# B&R Automation Studio project AcpTrakDemoTemplate
Automation Studio 4.10.3.60 SP; technology packages: mapp 5.18.0, mappControl 5.18.0, mappMotion 5.18.0, mappView 5.18.0

## Configuration Config1

CPU X20CP1685, AutomationRuntime G4.90, Build 4.1.2, Safety 0.0, Vc V4.72.2

### Task classes (Cpu.sw)
```
Cyclic#1 (cycle 800 us, tolerance 0 us):
  TrakCtrl <- Source.TrakCtrl.prg
Cyclic#4:
  MappCtrl <- Source.Infrastructure.MappCtrl.prg
Cyclic#8 (cycle 96000 us, tolerance 29952000 us):
  TrakProduc <- Source.Infrastructure.TrakProduction.prg
  TrakSvg <- Source.Infrastructure.TrakSvg.prg
DataObjects: McAcpSys
NcDataObjects: McDriveLog
Binaries: arsvcreg, udbdef, McAcpDrv, arflatprv, McProfGen, arcoal, TCData, FWRules, McAcpSim, mvLoader, ashwd, Config_1, ashwac, User, sysconf, asfw, arconfig, Config_3, Config_2, iomap, Role, Config_4, Config
Libraries: McBase, McAxis, McAcpTrak, MpBase, operator, runtime, astime, AsIecCon, AsBrStr, AsIODiag, sys_lib, standard, MTData, brsystem, MTTypes, MpAlarmX, MpServer, powerlnk, fileio, arssl, dataobj, aruser
```

### Hardware
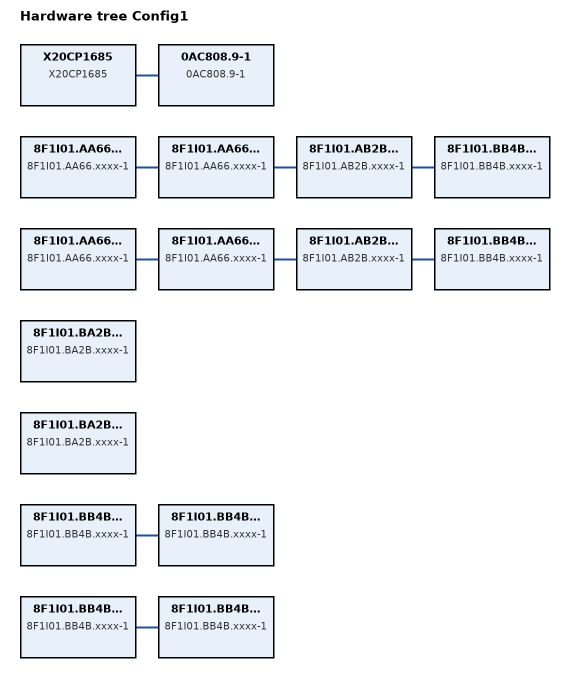
```
0AC808.9-1 : 0AC808.9-1 v1.0.0.0  [ETH1 -> X20CP1685.IF3 [Cable Type=PowerlinkCable, Length=10, Version=1.0.0.3]; ETH5 -> 8F1I01.BB4B.xxxx-1d.PLK3 [Cable Type=PowerlinkCable, Length=10, Version=1.0.0.3]; ETH8 -> 8F1I01.BB4B.xxxx-1e.PLK3 [Cable Type=PowerlinkCable, Length=10, Version=1.0.0.3]]
8F1I01.AA66.xxxx-1 : 8F1I01.AA66.xxxx-1 v1.0.0.2  [PLK1 -> 8F1I01.BA2B.xxxx-1c.PLK2 [Cable Type=PowerlinkCable, Length=10, Version=1.0.0.3]; PLK2 -> 8F1I01.AA66.xxxx-1e.PLK1 [Cable Type=PowerlinkCable, Length=10, Version=1.0.0.3]]
  EnableDNA = on
  DriveConfiguration:
    McTypeID = LLMConfig
  DriveConfiguration/Segment:
    Shape = STRAIGHT660
    SegmentReference = Seg_A_1
    SegmentSectorDirection = Positive
    ElongationCompensation = UseAssemblySetting
    StopReaction = UseAssemblySetting
    SpeedFilter = UseAssemblySetting
8F1I01.AA66.xxxx-1e : 8F1I01.AA66.xxxx-1 v1.0.0.2  [PLK1 -> 8F1I01.AA66.xxxx-1.PLK2 [Cable Type=PowerlinkCable, Length=10, Version=1.0.0.3]; PLK2 -> 8F1I01.AB2B.xxxx-1a.PLK1 [Cable Type=PowerlinkCable, Length=10, Version=1.0.0.3]]
  EnableDNA = on
  DriveConfiguration:
    McTypeID = LLMConfig
  DriveConfiguration/Segment:
    Shape = STRAIGHT660
    SegmentReference = Seg_A_2
    SegmentSectorDirection = Positive
    ElongationCompensation = UseAssemblySetting
    StopReaction = UseAssemblySetting
    SpeedFilter = UseAssemblySetting
8F1I01.AA66.xxxx-1f : 8F1I01.AA66.xxxx-1 v1.0.0.2  [PLK1 -> 8F1I01.BA2B.xxxx-1b.PLK2 [Cable Type=PowerlinkCable, Length=10, Version=1.0.0.3]; PLK2 -> 8F1I01.AA66.xxxx-1k.PLK1 [Cable Type=PowerlinkCable, Length=10, Version=1.0.0.3]]
  EnableDNA = on
  DriveConfiguration:
    McTypeID = LLMConfig
  DriveConfiguration/Segment:
    Shape = STRAIGHT660
    SegmentReference = Seg_A_8
    SegmentSectorDirection = Positive
    ElongationCompensation = UseAssemblySetting
    StopReaction = UseAssemblySetting
    SpeedFilter = UseAssemblySetting
8F1I01.AA66.xxxx-1k : 8F1I01.AA66.xxxx-1 v1.0.0.2  [PLK1 -> 8F1I01.AA66.xxxx-1f.PLK2 [Cable Type=PowerlinkCable, Length=10, Version=1.0.0.3]; PLK2 -> 8F1I01.AB2B.xxxx-1.PLK1 [Cable Type=PowerlinkCable, Length=10, Version=1.0.0.3]]
  EnableDNA = on
  DriveConfiguration:
    McTypeID = LLMConfig
  DriveConfiguration/Segment:
    Shape = STRAIGHT660
    SegmentReference = Seg_A_9
    SegmentSectorDirection = Positive
    ElongationCompensation = UseAssemblySetting
    StopReaction = UseAssemblySetting
    SpeedFilter = UseAssemblySetting
8F1I01.AB2B.xxxx-1 : 8F1I01.AB2B.xxxx-1 v1.0.0.2  [PLK1 -> 8F1I01.AA66.xxxx-1k.PLK2 [Cable Type=PowerlinkCable, Length=10, Version=1.0.0.3]; PLK2 -> 8F1I01.BB4B.xxxx-1.PLK1 [Cable Type=PowerlinkCable, Length=10, Version=1.0.0.3]]
  EnableDNA = on
  DriveConfiguration:
    McTypeID = LLMConfig
  DriveConfiguration/Segment:
    Shape = STRAIGHT105_TO_CIRCULAR
    SegmentReference = Seg_A_10
    SegmentSectorDirection = Positive
    ElongationCompensation = UseAssemblySetting
    StopReaction = UseAssemblySetting
    SpeedFilter = UseAssemblySetting
8F1I01.AB2B.xxxx-1a : 8F1I01.AB2B.xxxx-1 v1.0.0.2  [PLK1 -> 8F1I01.AA66.xxxx-1e.PLK2 [Cable Type=PowerlinkCable, Length=10, Version=1.0.0.3]; PLK2 -> 8F1I01.BB4B.xxxx-1b.PLK1 [Cable Type=PowerlinkCable, Length=10, Version=1.0.0.3]]
  EnableDNA = on
  DriveConfiguration:
    McTypeID = LLMConfig
  DriveConfiguration/Segment:
    Shape = STRAIGHT105_TO_CIRCULAR
    SegmentReference = Seg_A_3
    SegmentSectorDirection = Positive
    ElongationCompensation = UseAssemblySetting
    StopReaction = UseAssemblySetting
    SpeedFilter = UseAssemblySetting
8F1I01.BA2B.xxxx-1b : 8F1I01.BA2B.xxxx-1 v1.0.0.2  [PLK1 -> 8F1I01.BB4B.xxxx-1c.PLK2 [Cable Type=PowerlinkCable, Length=10, Version=1.0.0.3]; PLK2 -> 8F1I01.AA66.xxxx-1f.PLK1 [Cable Type=PowerlinkCable, Length=10, Version=1.0.0.3]]
  EnableDNA = on
  DriveConfiguration:
    McTypeID = LLMConfig
  DriveConfiguration/Segment:
    Shape = CIRCULAR_TO_STRAIGHT105
    SegmentReference = Seg_A_7
    SegmentSectorDirection = Positive
    ElongationCompensation = UseAssemblySetting
    StopReaction = UseAssemblySetting
    SpeedFilter = UseAssemblySetting
8F1I01.BA2B.xxxx-1c : 8F1I01.BA2B.xxxx-1 v1.0.0.2  [PLK1 -> 8F1I01.BB4B.xxxx-1a.PLK2 [Cable Type=PowerlinkCable, Length=10, Version=1.0.0.3]; PLK2 -> 8F1I01.AA66.xxxx-1.PLK1 [Cable Type=PowerlinkCable, Length=10, Version=1.0.0.3]]
  EnableDNA = on
  DriveConfiguration:
    McTypeID = LLMConfig
  DriveConfiguration/Segment:
    Shape = CIRCULAR_TO_STRAIGHT105
    SegmentReference = Seg_A_14
    SegmentSectorDirection = Positive
    ElongationCompensation = UseAssemblySetting
    StopReaction = UseAssemblySetting
    SpeedFilter = UseAssemblySetting
8F1I01.BB4B.xxxx-1 : 8F1I01.BB4B.xxxx-1 v1.0.0.2  [PLK1 -> 8F1I01.AB2B.xxxx-1.PLK2 [Cable Type=PowerlinkCable, Length=10, Version=1.0.0.3]]
  EnableDNA = on
  DriveConfiguration:
    McTypeID = LLMConfig
  DriveConfiguration/Segment:
    Shape = CIRCULAR
    SegmentReference = Seg_A_11
    SegmentSectorDirection = Positive
    ElongationCompensation = UseAssemblySetting
    StopReaction = UseAssemblySetting
    SpeedFilter = UseAssemblySetting
8F1I01.BB4B.xxxx-1a : 8F1I01.BB4B.xxxx-1 v1.0.0.2  [PLK1 -> 8F1I01.BB4B.xxxx-1d.PLK2 [Cable Type=PowerlinkCable, Length=10, Version=1.0.0.3]; PLK2 -> 8F1I01.BA2B.xxxx-1c.PLK1 [Cable Type=PowerlinkCable, Length=10, Version=1.0.0.3]]
  EnableDNA = on
  DriveConfiguration:
    McTypeID = LLMConfig
  DriveConfiguration/Segment:
    Shape = CIRCULAR
    SegmentReference = Seg_A_13
    SegmentSectorDirection = Positive
    ElongationCompensation = UseAssemblySetting
    StopReaction = UseAssemblySetting
    SpeedFilter = UseAssemblySetting
8F1I01.BB4B.xxxx-1b : 8F1I01.BB4B.xxxx-1 v1.0.0.2  [PLK1 -> 8F1I01.AB2B.xxxx-1a.PLK2 [Cable Type=PowerlinkCable, Length=10, Version=1.0.0.3]]
  EnableDNA = on
  DriveConfiguration:
    McTypeID = LLMConfig
  DriveConfiguration/Segment:
    Shape = CIRCULAR
    SegmentReference = Seg_A_4
    SegmentSectorDirection = Positive
    ElongationCompensation = UseAssemblySetting
    StopReaction = UseAssemblySetting
    SpeedFilter = UseAssemblySetting
8F1I01.BB4B.xxxx-1c : 8F1I01.BB4B.xxxx-1 v1.0.0.2  [PLK1 -> 8F1I01.BB4B.xxxx-1e.PLK2 [Cable Type=PowerlinkCable, Length=10, Version=1.0.0.3]; PLK2 -> 8F1I01.BA2B.xxxx-1b.PLK1 [Cable Type=PowerlinkCable, Length=10, Version=1.0.0.3]]
  EnableDNA = on
  DriveConfiguration:
    McTypeID = LLMConfig
  DriveConfiguration/Segment:
    Shape = CIRCULAR
    SegmentReference = Seg_A_6
    SegmentSectorDirection = Positive
    ElongationCompensation = UseAssemblySetting
    StopReaction = UseAssemblySetting
    SpeedFilter = UseAssemblySetting
8F1I01.BB4B.xxxx-1d : 8F1I01.BB4B.xxxx-1 v1.0.0.2  [PLK2 -> 8F1I01.BB4B.xxxx-1a.PLK1 [Cable Type=PowerlinkCable, Length=10, Version=1.0.0.3]; PLK3 -> 0AC808.9-1.ETH5 [Cable Type=PowerlinkCable, Length=10, Version=1.0.0.3]]
  EnableDNA = on
  DriveConfiguration:
    McTypeID = LLMConfig
  DriveConfiguration/Segment:
    Shape = CIRCULAR
    SegmentReference = Seg_A_12
    SegmentSectorDirection = Positive
    ElongationCompensation = UseAssemblySetting
    StopReaction = UseAssemblySetting
    SpeedFilter = UseAssemblySetting
8F1I01.BB4B.xxxx-1e : 8F1I01.BB4B.xxxx-1 v1.0.0.2  [PLK2 -> 8F1I01.BB4B.xxxx-1c.PLK1 [Cable Type=PowerlinkCable, Length=10, Version=1.0.0.3]; PLK3 -> 0AC808.9-1.ETH8 [Cable Type=PowerlinkCable, Length=10, Version=1.0.0.3]]
  EnableDNA = on
  DriveConfiguration:
    McTypeID = LLMConfig
  DriveConfiguration/Segment:
    Shape = CIRCULAR
    SegmentReference = Seg_A_5
    SegmentSectorDirection = Positive
    ElongationCompensation = UseAssemblySetting
    StopReaction = UseAssemblySetting
    SpeedFilter = UseAssemblySetting
X20CP1685 : X20CP1685 v1.4.0.0
  Connector IF2:
    ActivateDevice = 1
  Connector IF3:
    CycleTime = 800
  ConfigurationID = AcpTrakVolpak_Config1
  Simulation = 1
  TimerDeviceType = EPLX2X
  TimerDevice = X20CP1685.IF3
  TaskClassIdleTime = 800
  Cyclic1Duration = 800
  Cyclic1Tolerance = 0
  Cyclic3Duration = 49600
  Cyclic3Tolerance = 49600
  Cyclic8Duration = 96000
  Cyclic8Tolerance = 29952000
  FileDevice1
  FileDeviceName1 = SvgData
  FileDevicePath1 = C:\DataTrak\
  ActivateOpcUa = 1
  OpcUaInformationModels_PV_Version = 1
```

### Config_1.assembly - X20CP1685/mappMotion/TrakOval/Config_1.assembly
```
Element gAssembly_1 (Type=assembly)
  Tracks:
    TrackSeparation = 0.030
    Track[1]:
      Segments:
        SegmentRef[1] = ::Seg_A_1
        SegmentRef[2] = ::Seg_A_2
        SegmentRef[3] = ::Seg_A_3
        SegmentRef[4] = ::Seg_A_4
        SegmentRef[5] = ::Seg_A_5
        SegmentRef[6] = ::Seg_A_6
        SegmentRef[7] = ::Seg_A_7
        SegmentRef[8] = ::Seg_A_8
        SegmentRef[9] = ::Seg_A_9
        SegmentRef[10] = ::Seg_A_10
        SegmentRef[11] = ::Seg_A_11
        SegmentRef[12] = ::Seg_A_12
        SegmentRef[13] = ::Seg_A_13
        SegmentRef[14] = ::Seg_A_14
      Position = Absolute
        SegmentRef = ::Seg_A_1
        SegmentCountDirection = RightToLeft
        Translation:
          X = 0.0
          Y = 0.0
          Z = 0.0
        Orientation:
          Angle1 = 0.0
          Angle2 = 180.0
          Angle3 = 0.0
  CommonSegmentSettings:
    SegmentSimulationOnPLC = Off
    ElongationCompensation = Inactive
    StopReaction = InductionHalt
    SpeedFilter = Lowpass
      FilterTime = 0.0008
    ControllerParameters:
      DefaultParameter:
        Controller:
          Position:
            ProportionalGain = 200
          Speed:
            ProportionalGain = 80
            IntegrationTime = 0.0
          FeedForward:
            TotalMass = 1.0
            ForcePositive = 1.5
            ForceNegative = 1.5
            SpeedForceFactor = 1.4
            ForceLoad = 0.0
        MovementErrorLimits:
          PositionError = 0.01
          VelocityError = 50
        Diverter:
          ForceOverride = 1.0
      AdditionalParameterSets = NotUsed
    ScopeOfErrorReaction = Assembly
    ShuttleIdentificationTime = 0
  Shuttles:
    MaxShuttleCount = 100
    MaxShuttleCommandCount = 0
    UseConvoys = Active
    DistanceReserve:
      Collision = 0.002
      ErrorStop = 0.006
    ShuttleStereotypes:
      ShuttleStRef[1] = ShuttleStereotype_1
    MagnetPlateConfigurations:
      ShuttleType[1] = 8F1SA.102.xxxxxx-x
    CollisionAvoidance:
      Strategy = Constant
      MaximumModelDimensions:
        Length:
          ExtentToFront = 0.025
          ExtentToBack = 0.025
        Width:
          Width = 0.046
  Visualization:
    MonitoringPv = 
    ProcessingTaskClass = 4
  Alarms = MpAlarmX
```

### Config_2.shuttlestereotype - X20CP1685/mappMotion/TrakOval/Config_2.shuttlestereotype
```
Element ShuttleStereotype_1 (Type=shuttlestereotype)
  MeasurementUnit = 5067858
  MeasurementResolution = 0.00001
  MovementLimits = Internal
    VelocityIsReadOnly = 0
    Velocity:
      Velocity = 4.0
    AccelerationIsReadOnly = 0
    Acceleration:
      Acceleration = 40.0
    DecelerationIsReadOnly = 0
    Deceleration:
      Deceleration = 40.0
    UpdateMode = Immediately
  JerkFilter = NotUsed
  UserData:
    Size = 52
  StateTransitions:
    AutomaticRecontrol = Active
```

### Config_3.sector - X20CP1685/mappMotion/TrakOval/Config_3.sector
```
Element SectorTrackA (Type=sector)
  Type = Composed
    StartSegment:
      SegmentRef = ::Seg_A_1
    IntermediateSegments:
      SegmentRef[1] = ::Seg_A_1
      SegmentRef[2] = ::Seg_A_2
      SegmentRef[3] = ::Seg_A_3
      SegmentRef[4] = ::Seg_A_4
      SegmentRef[5] = ::Seg_A_5
      SegmentRef[6] = ::Seg_A_6
      SegmentRef[7] = ::Seg_A_7
      SegmentRef[8] = ::Seg_A_8
      SegmentRef[9] = ::Seg_A_9
      SegmentRef[10] = ::Seg_A_10
      SegmentRef[11] = ::Seg_A_11
      SegmentRef[12] = ::Seg_A_12
      SegmentRef[13] = ::Seg_A_13
    EndSegment:
      SegmentRef = ::Seg_A_14
      PositionRelativeTo = FromEnd
  Alarms = MpAlarmX
```

### Config_4.processpointlist - X20CP1685/mappMotion/TrakOval/Config_4.processpointlist
```
Element ProcessPointList_Template (Type=processpointlist)
  ProcessPoint[0]:
    Name = PP_Test
    SectorRef = SectorTrackA
    TriggerEventBufferSize = 10
    BarrierFunctionality = Off
Element ProcessPointList_Machine (Type=processpointlist)
  ProcessPoint[0]:
    Name = PP_Init
    SectorRef = SectorTrackA
    TriggerEventBufferSize = 10
    BarrierFunctionality = On
  ProcessPoint[1]:
    Name = PP_Stop
    SectorRef = SectorTrackA
    Position = 1.5
    TriggerEventBufferSize = 10
    BarrierFunctionality = On
  ProcessPoint[2]:
    Name = PP_Stop1
    SectorRef = SectorTrackA
    Position = 3
    TriggerEventBufferSize = 10
    BarrierFunctionality = On
```

### Config_5.mappmotioncfg - X20CP1685/mappMotion/TrakOval/Config_5.mappmotioncfg
```
Element MappMotionConfiguration (Type=mappmotioncfg)
  Processing:
    ProcessingTaskClass = 1
  SharedAlarms:
    Axis = MpAlarmX
    Segment = MpAlarmX
    Sector = MpAlarmX
    Shuttle = MpAlarmX
      mapp.AlarmX.Core.Configuration:
        [3]:
          AdditionalInformation1 = Shuttle
```

## Logical view

Binary libraries used (declarations not repeated): operator, runtime, astime, AsIecCon, AsBrStr, AsIODiag, sys_lib, standard, McBase, McAcpTrak, McAxis, MpBase, MTData 5.18.0, brsystem, MTTypes, MpAlarmX, MpServer

### Global.var
```iecst
VAR
	Seg_A_1 : McSegmentType;
	Seg_A_2 : McSegmentType;
	Seg_A_3 : McSegmentType;
	Seg_A_4 : McSegmentType;
	Seg_A_5 : McSegmentType;
	Seg_A_6 : McSegmentType;
	Seg_A_7 : McSegmentType;
	Seg_A_8 : McSegmentType;
	Seg_A_9 : McSegmentType;
	Seg_A_10 : McSegmentType;
	Seg_A_11 : McSegmentType;
	Seg_A_12 : McSegmentType;
	Seg_A_13 : McSegmentType;
	Seg_A_14 : McSegmentType;
END_VAR
```

### gTrak.typ - Global data types
```iecst
(*interface assembly control*)

TYPE
	TrakAsmType : 	STRUCT
		AssemblyRef : REFERENCE TO McAssemblyType; (*assembly reference - ADR(gAssembly_1)*)
		CmdPower : BOOL; (*command power on/off*)
		CmdErrorReset : BOOL; (*command error reset*)
		CmdAllShuttleMoveStop : BOOL;
		CmdAllShuttleMovePosition : BOOL;
		CmdAllShuttleMoveVelocity : BOOL;
		StatusSimulated : BOOL; (*status assembly is simulated*)
		StatusDisabled : BOOL; (*status assembly is disabled*)
		StatusReady : BOOL; (*status assembly is ready*)
		StatusHoming : BOOL; (*status assembly is homing*)
		StatusStopping : BOOL; (*status assembly is stopping*)
		StatusErrorStop : BOOL; (*status assembly is in error-stop*)
		StatusCommunicationReady : BOOL; (*status PLK communication to all segments in assembly is ready*)
		StatusReadyForPower : BOOL; (*status assembly is ready for command power-on*)
		StatusPower : BOOL; (*status assembly is power-on*)
		StatusReadyForMovement : BOOL; (*status assembly is ready to start shuttle movements*)
		MonitorSegmentsPresent : UINT; (*monitor segment present on assembly*)
		MonitorSegmentsInErrorStop : UINT; (*monitor segment in error-stop*)
		MonitorShuttlesPresent : UINT; (*monitor shuttles present on assembly*)
		MonitorShuttlesInErrorStop : UINT; (*monitor shuttles in error-stop*)
		ParaMoveSectorRef : REFERENCE TO McSectorType; (*parameter shuttle move target sector - ADR(Sector_x)*)
		ParaMovePosition : LREAL; (*parameter shuttle move target position*)
		ParaMoveVelocity : REAL; (*parameter shuttle move target velocity*)
		ParaMoveRouteVelocity : REAL; (*parameter shuttle move routing velocity*)
		ParaMoveAcceleration : REAL; (*parameter shuttle move acceleration*)
		ParaMoveDeceleration : REAL; (*parameter shuttle move deceleration*)
		Segment : ARRAY[1..TRAK_MAX_SEGMENT]OF TrakAsmSegmentType;
		Shuttle : ARRAY[1..TRAK_MAX_SHUTTLE]OF TrakAsmShuttleType; (*shuttle information*)
	END_STRUCT;
	TrakAsmShuttleType : 	STRUCT
		Valid : BOOL; (*shuttledata valid*)
		Axis : McAxisType; (*McAxis of shuttle*)
		ID : UDINT; (*shuttle ID as displayed in logger and SceneViewer - TODO*)
		ActSectorType : McAcpTrakSecTypeEnum; (*shuttle current sector type*)
		ActSector : STRING[32]; (*shuttle current sector*)
		ActPosition : LREAL; (*shuttle position on sector*)
		ActVelocity : REAL; (*shuttle velocity on sector*)
		TotalMoveDistance : LREAL; (*shuttle total moved distance*)
		StatusStandStill : BOOL; (*shuttle is in state Standstill*)
		StatusStopping : BOOL; (*shuttle is in state Stopping*)
		StatusErrorStop : BOOL; (*shuttle is in state Errorstop*)
		StatusDiscreteMotion : BOOL; (*shuttle is in state DiscreteMotion*)
		StatusContinuousMotion : BOOL; (*shuttle is in state ContinuousMotion*)
		StatusSynchronizedMotion : BOOL; (*shuttle is in state SynchronizedMotion*)
	END_STRUCT;
	TrakAsmSegmentType : 	STRUCT
		Valid : BOOL;
		Segment : McSegmentType;
		StatusDisabled : BOOL;
		StatusReady : BOOL;
		StatusStopping : BOOL;
		StatusErrorStop : BOOL;
		StatusShuttlesInError : BOOL;
	END_STRUCT;
END_TYPE

(*shuttle UserData structure - adapt to your application*)

TYPE
	TrakShuttleUserDataType : 	STRUCT
		SceneColorRed : REAL; (*do not change: SceneViewer shuttle colour red*)
		SceneColorGreen : REAL; (*do not change: SceneViewer shuttle colour green*)
		SceneColorBlue : REAL; (*do not change: SceneViewer shuttle colour blue*)
		SceneText : STRING[31]; (*do not change: SceneViewer shuttle text*)
		Test : USINT; (*do not change: for use in TrakTest task*)
		ID : UINT; (*shuttle ID*)
		InitDone : BOOL; (*example: product weight*)
	END_STRUCT;
END_TYPE
```

### gTrak.var - Global variables
```iecst
(*interface assembly control*)
VAR
	gTrakAsm : TrakAsmType; (*trak assembly main interface structure*)
END_VAR
(*production control*)
VAR
	gProducedProduct : UINT; (*number of produced products (in ppm)*)
END_VAR
(*constants*)
VAR CONSTANT
	TRAK_MAX_SHUTTLE : UINT := 72; (*maximum number of shuttles handled in this application - should be set equal or higher than Shuttles-maximum-count setting in mappMotion assembly config file*)
	TRAK_MAX_SEGMENT : UINT := 24; (*maximum number of segments handled in this application*)
END_VAR
```

### Program Logical/Source/TrakCtrl (IEC) - trak assembly control

#### Types.typ
```iecst
(*enum*)

TYPE
	TrakSimShuttleType : 	STRUCT
		SectorRef : REFERENCE TO McSectorType; (*add shuttle in simulation at sector - ADR(Sector_x)*)
		Position : LREAL; (*add shuttle in simulation at position*)
	END_STRUCT;
	StepEnum :
		(
		COMMAND := 0,
		RESET,
		ASM_POWER_ON := 10,
		ASM_POWER_ON_WAIT,
		GET_SEGMENT_INIT := 20,
		GET_SEGMENT,
		GET_SEGMENT_WAIT,
		ADD_SHUTTLE_INIT := 30,
		ADD_SHUTTLE,
		ADD_SHUTTLE_WAIT,
		GET_SHUTTLE_INIT := 40,
		GET_SHUTTLE,
		GET_SHUTTLE_WAIT,
		ERROR := 99,
		READY := 100,
		ASM_POWER_OFF := 110,
		ASM_POWER_OFF_WAIT,
		ASM_SH_DELETE,
		ASM_SH_DELETE_WAIT,
		STOP_SHUTTLE := 120,
		STOP_SHUTTLE_WAIT,
		MOVE_SHUTTLE_VELOCITY := 130,
		MOVE_SHUTTLE_VELOCITY_WAIT,
		MOVE_SHUTTLE_POSITION := 140,
		MOVE_SHUTTLE_POSITION_WAIT
		);
END_TYPE
```

#### Variables.var
```iecst
(*sequence control*)
VAR
	Step : StepEnum;
	i : UINT;
	CntShuttle : UINT;
	CntSegment : UINT;
END_VAR
(*add shuttles for simulation*)
VAR
	SimNumShuttle : USINT := 4;
	SimShuttle : ARRAY[1..TRAK_MAX_SHUTTLE] OF TrakSimShuttleType;
END_VAR
(*initialze shuttle user data*)
VAR
	SizeofShuttleUserData : UDINT;
	ShuttleUserData : TrakShuttleUserDataType;
END_VAR
(*assembly FUB*)
VAR
	MC_BR_AsmReset_AcpTrak_0 : MC_BR_AsmReset_AcpTrak;
	MC_BR_AsmPowerOn_AcpTrak_0 : MC_BR_AsmPowerOn_AcpTrak;
	MC_BR_AsmPowerOff_AcpTrak_0 : MC_BR_AsmPowerOff_AcpTrak;
	MC_BR_AsmGetInfo_AcpTrak_0 : MC_BR_AsmGetInfo_AcpTrak;
	MC_BR_AsmReadStatus_AcpTrak_0 : MC_BR_AsmReadStatus_AcpTrak;
	MC_BR_AsmReadInfo_AcpTrak_0 : MC_BR_AsmReadInfo_AcpTrak;
	MC_BR_AsmGetSegment_AcpTrak_0 : MC_BR_AsmGetSegment_AcpTrak;
	MC_BR_SecAddShuttle_AcpTrak_0 : MC_BR_SecAddShuttle_AcpTrak;
	MC_BR_AsmGetShuttle_AcpTrak_0 : MC_BR_AsmGetShuttle_AcpTrak;
	MC_BR_AsmDeleteShuttle_AcpTrak_0 : MC_BR_AsmDeleteShuttle_AcpTrak;
END_VAR
(*segment FUB*)
VAR
	MC_BR_SegReadStatus_AcpTrak_0 : ARRAY[1..TRAK_MAX_SEGMENT] OF MC_BR_SegReadStatus_AcpTrak;
END_VAR
(*shuttle FUB*)
VAR
	MC_BR_ShCopyUserData_AcpTrak_0 : MC_BR_ShCopyUserData_AcpTrak;
	MC_BR_ShReadInfo_AcpTrak_0 : ARRAY[1..TRAK_MAX_SHUTTLE] OF MC_BR_ShReadInfo_AcpTrak;
	MC_ReadStatus_0 : ARRAY[1..TRAK_MAX_SHUTTLE] OF MC_ReadStatus;
	MC_Stop_0 : MC_Stop;
	MC_BR_RoutedMoveVel_AcpTrak_0 : MC_BR_RoutedMoveVel_AcpTrak;
	MC_BR_RoutedMoveAbs_AcpTrak_0 : MC_BR_RoutedMoveAbs_AcpTrak;
END_VAR
```

#### Main.st
```iecst
//////////////////////////////////////////////////////////////////////////////////////////////////////////////////////////////
//
// Copyright B&R Industrial Automation GmbH
// Author    B&R
// Created   Feb 1, 2018
//
// trak assembly basic control task
// TC#1 => preferred to be attached to mappMotion task class
//
// * assembly startup sequence
// * ErrorStop handling
// * basic shuttle handling
// * aggregated shuttle move commands
//
// "gTrakAsm" - global interface structure
//
//////////////////////////////////////////////////////////////////////////////////////////////////////////////////////////////

PROGRAM _INIT

	//////////////////////////////////////////////////////////////////////////////////////////////////////////////////////////////
	// interface structure

	gTrakAsm.AssemblyRef				:= ADR(gAssembly_1);
	gTrakAsm.CmdPower					:= FALSE;
	gTrakAsm.CmdErrorReset				:= FALSE;

	gTrakAsm.CmdAllShuttleMoveStop		:= FALSE;
	gTrakAsm.CmdAllShuttleMovePosition	:= FALSE;
	gTrakAsm.CmdAllShuttleMoveVelocity	:= FALSE;
	gTrakAsm.ParaMoveSectorRef			:= ADR(SectorTrackA);
	gTrakAsm.ParaMovePosition			:= 2.0;
	gTrakAsm.ParaMoveVelocity			:= 2.0;
	gTrakAsm.ParaMoveRouteVelocity		:= 2.0;
	gTrakAsm.ParaMoveAcceleration		:= 20.0;
	gTrakAsm.ParaMoveDeceleration		:= 20.0;

	Step := COMMAND;

	// size of ShuttleUserData structure - this value has to be entered in ShuttleStereotype -> UserData -> Size
	SizeofShuttleUserData := SIZEOF(ShuttleUserData);

END_PROGRAM

PROGRAM _CYCLIC

	//////////////////////////////////////////////////////////////////////////////////////////////////////////////////////////////
	// global ErrorStop and ErrorReset
	IF(gTrakAsm.StatusErrorStop)THEN
		gTrakAsm.StatusReadyForMovement := FALSE;
		Step := ERROR;
	END_IF
	IF(gTrakAsm.CmdErrorReset)THEN
		gTrakAsm.CmdErrorReset := FALSE;
		MC_BR_AsmReset_AcpTrak_0.Execute := TRUE;
	END_IF

	CASE Step OF

		//////////////////////////////////////////////////////////////////////////////////////////////////////////////////////////////
		// command
		COMMAND:
			IF(gTrakAsm.CmdPower)THEN
				Step := RESET;
			END_IF

		//////////////////////////////////////////////////////////////////////////////////////////////////////////////////////////////
		// startup sequence

		// reset
		RESET:

			brsmemset(ADR(gTrakAsm.Segment), 0, SIZEOF(gTrakAsm.Segment));
			brsmemset(ADR(gTrakAsm.Shuttle), 0, SIZEOF(gTrakAsm.Shuttle));

			MC_BR_AsmGetSegment_AcpTrak_0.Enable := FALSE;
			MC_BR_AsmGetShuttle_AcpTrak_0.Enable := FALSE;

			Step := ASM_POWER_ON;

		// assembly power ON
		ASM_POWER_ON:

			IF(gTrakAsm.StatusDisabled)THEN
				MC_BR_AsmPowerOn_AcpTrak_0.Execute := TRUE;
			END_IF
			Step := ASM_POWER_ON_WAIT;

		ASM_POWER_ON_WAIT:

			IF(gTrakAsm.StatusReady)THEN
				Step := GET_SEGMENT_INIT;
			END_IF

		GET_SEGMENT_INIT:

			MC_BR_AsmGetSegment_AcpTrak_0.Enable 	:= TRUE;
			MC_BR_AsmGetSegment_AcpTrak_0.Next 		:= FALSE;
			CntSegment 	:= 0;
			Step 		:= GET_SEGMENT_WAIT;

		GET_SEGMENT:

			MC_BR_AsmGetSegment_AcpTrak_0.Next := TRUE;
			Step := GET_SEGMENT_WAIT;

		GET_SEGMENT_WAIT:

			IF(MC_BR_AsmGetSegment_AcpTrak_0.Error)THEN
				MC_BR_AsmGetSegment_AcpTrak_0.Enable := FALSE;
				Step := ERROR;

			ELSIF (MC_BR_AsmGetSegment_AcpTrak_0.Valid) THEN

				gTrakAsm.MonitorSegmentsPresent := MC_BR_AsmGetSegment_AcpTrak_0.TotalCount;

				IF(MC_BR_AsmGetSegment_AcpTrak_0.TotalCount = 0)THEN	// no segments present present
					MC_BR_AsmGetSegment_AcpTrak_0.Enable := FALSE;
					Step := ERROR;
				ELSE

					CntSegment := CntSegment + 1;
					gTrakAsm.Segment[CntSegment].Segment := MC_BR_AsmGetSegment_AcpTrak_0.Segment;

					IF(MC_BR_AsmGetSegment_AcpTrak_0.RemainingCount = 0)THEN	// all present segments read => ok, proceed
						MC_BR_AsmGetSegment_AcpTrak_0.Enable := FALSE;
						Step := ADD_SHUTTLE_INIT;
					ELSIF(CntSegment >= TRAK_MAX_SEGMENT)THEN					// more segments present than max configured => error
						MC_BR_AsmGetSegment_AcpTrak_0.Enable := FALSE;
						Step := ERROR;
					ELSE														// read next => positive edge on .Next flag
						MC_BR_AsmGetSegment_AcpTrak_0.Next := FALSE;
						Step := GET_SEGMENT;
					END_IF
				END_IF

			END_IF

		// add shuttles (for simulation only)
		ADD_SHUTTLE_INIT:

			IF(gTrakAsm.StatusSimulated)THEN
				// Define the simulated position for each shuttle
				FOR i:=1 TO TRAK_MAX_SHUTTLE DO
					IF ((i < SimNumShuttle) AND (SimNumShuttle <= TRAK_MAX_SHUTTLE)) THEN
						SimShuttle[i].SectorRef := ADR(SectorTrackA);
						SimShuttle[i].Position 	:= 0.355 + UINT_TO_LREAL(SimNumShuttle - i)/10.0;
					ELSE
						SimShuttle[i].SectorRef := ADR(SectorTrackA);
						SimShuttle[i].Position 	:= 0.355;
					END_IF
				END_FOR
				CntShuttle 	:= 0;
				Step 		:= ADD_SHUTTLE;
			ELSE
				Step := GET_SHUTTLE_INIT;
			END_IF

		ADD_SHUTTLE:

			CntShuttle := CntShuttle + 1;
			IF(CntShuttle > SimNumShuttle)THEN
				Step := GET_SHUTTLE_INIT;
			ELSIF(SimShuttle[CntShuttle].SectorRef = 0)THEN
				Step := GET_SHUTTLE_INIT;
			ELSE
				MC_BR_SecAddShuttle_AcpTrak_0.Sector		:= SimShuttle[CntShuttle].SectorRef;
				MC_BR_SecAddShuttle_AcpTrak_0.Execute		:= TRUE;
				MC_BR_SecAddShuttle_AcpTrak_0.Position		:= SimShuttle[CntShuttle].Position;
				MC_BR_SecAddShuttle_AcpTrak_0.AdvancedParameters.Velocity		:= 0.0;
				MC_BR_SecAddShuttle_AcpTrak_0.AdvancedParameters.Orientation	:= mcDIR_POSITIVE;
				Step := ADD_SHUTTLE_WAIT;
			END_IF

		ADD_SHUTTLE_WAIT:
			IF(MC_BR_SecAddShuttle_AcpTrak_0.Error)THEN
				Step := ERROR;

			ELSIF(MC_BR_SecAddShuttle_AcpTrak_0.Done)THEN
				Step := ADD_SHUTTLE;
			END_IF

		// get all shuttles present on assembly
		GET_SHUTTLE_INIT:

			MC_BR_AsmGetShuttle_AcpTrak_0.Enable 	:= TRUE;
			MC_BR_AsmGetShuttle_AcpTrak_0.Next 		:= FALSE;
			CntShuttle 	:= 0;
			Step 		:= GET_SHUTTLE_WAIT;

		GET_SHUTTLE:

			MC_BR_AsmGetShuttle_AcpTrak_0.Next := TRUE;
			Step := GET_SHUTTLE_WAIT;

		GET_SHUTTLE_WAIT:

			IF(MC_BR_AsmGetShuttle_AcpTrak_0.Error)THEN
				MC_BR_AsmGetShuttle_AcpTrak_0.Enable := FALSE;
				Step := ERROR;

			ELSIF(MC_BR_AsmGetShuttle_AcpTrak_0.Valid)THEN
				gTrakAsm.MonitorShuttlesPresent := MC_BR_AsmGetShuttle_AcpTrak_0.TotalCount;

				IF(MC_BR_AsmGetShuttle_AcpTrak_0.TotalCount = 0)THEN			// no shuttles present => ok, proceed
					MC_BR_AsmGetShuttle_AcpTrak_0.Enable := FALSE;
					Step := READY;
				ELSE
					CntShuttle := CntShuttle + 1;
					gTrakAsm.Shuttle[CntShuttle].Axis	:= MC_BR_AsmGetShuttle_AcpTrak_0.Axis;
					gTrakAsm.Shuttle[CntShuttle].ID		:= MC_BR_AsmGetShuttle_AcpTrak_0.AdditionalInfo.ShuttleID;

					// initialize shuttle UserData (White colour)
					ShuttleUserData.SceneColorRed	:= 1.0;
					ShuttleUserData.SceneColorGreen	:= 1.0;
					ShuttleUserData.SceneColorBlue	:= 1.0;
					ShuttleUserData.ID				:= CntShuttle;

					MC_BR_ShCopyUserData_AcpTrak_0.Axis			:= ADR(gTrakAsm.Shuttle[CntShuttle].Axis);
					MC_BR_ShCopyUserData_AcpTrak_0.Execute		:= TRUE;
					MC_BR_ShCopyUserData_AcpTrak_0.DataAddress	:= ADR(ShuttleUserData);
					MC_BR_ShCopyUserData_AcpTrak_0.DataSize		:= SIZEOF(ShuttleUserData);
					MC_BR_ShCopyUserData_AcpTrak_0.Mode			:= mcACPTRAK_USERDATA_SET;

					IF(MC_BR_AsmGetShuttle_AcpTrak_0.RemainingCount = 0)THEN	// all present shuttles read => ok, proceed
						MC_BR_AsmGetShuttle_AcpTrak_0.Enable := FALSE;
						Step := READY;
					ELSIF(CntShuttle >= TRAK_MAX_SHUTTLE)THEN					// more shuttles present than max configured => error
						MC_BR_AsmGetShuttle_AcpTrak_0.Enable := FALSE;
						Step := ERROR;
					ELSE														// read next => positive edge on .Next flag
						MC_BR_AsmGetShuttle_AcpTrak_0.Next := FALSE;
						Step := GET_SHUTTLE;
					END_IF
				END_IF
			END_IF

		//////////////////////////////////////////////////////////////////////////////////////////////////////////////////////////////
		// assembly ErrorStop => ErrorReset required
		ERROR:

			gTrakAsm.CmdPower := FALSE;
			gTrakAsm.MonitorShuttlesPresent := 0;

			IF(gTrakAsm.StatusDisabled)THEN
				Step := COMMAND;
			ELSIF(gTrakAsm.StatusReady)THEN
				Step := ASM_POWER_OFF;
			END_IF

		//////////////////////////////////////////////////////////////////////////////////////////////////////////////////////////////
		// assembly Active and ready for movement
		READY:

			gTrakAsm.StatusReadyForMovement := TRUE;
			IF(gTrakAsm.CmdPower = 0)THEN
				gTrakAsm.StatusReadyForMovement := FALSE;
				Step := ASM_POWER_OFF;

			ELSIF(gTrakAsm.CmdAllShuttleMoveStop)THEN
				gTrakAsm.CmdAllShuttleMoveStop := 0;
				CntShuttle := 0;
				Step := STOP_SHUTTLE;

			ELSIF(gTrakAsm.CmdAllShuttleMoveVelocity)THEN
				gTrakAsm.CmdAllShuttleMoveVelocity := 0;
				CntShuttle := 0;
				Step := MOVE_SHUTTLE_VELOCITY;

			ELSIF(gTrakAsm.CmdAllShuttleMovePosition)THEN
				gTrakAsm.CmdAllShuttleMovePosition := 0;
				CntShuttle := 0;
				Step := MOVE_SHUTTLE_POSITION;
			END_IF

		//////////////////////////////////////////////////////////////////////////////////////////////////////////////////////////////
		// assembly power OFF
		ASM_POWER_OFF:
			MC_BR_AsmPowerOff_AcpTrak_0.Execute := TRUE;
			Step := ASM_POWER_OFF_WAIT;

		ASM_POWER_OFF_WAIT:
			IF(gTrakAsm.StatusDisabled)THEN
				gTrakAsm.MonitorShuttlesPresent := 0;
				Step := ASM_SH_DELETE;
			END_IF

		//////////////////////////////////////////////////////////////////////////////////////////////////////////////////////////////
		// delete assembly shuttles
		ASM_SH_DELETE:
			MC_BR_AsmDeleteShuttle_AcpTrak_0.Execute := TRUE;
			Step := ASM_SH_DELETE_WAIT;

		ASM_SH_DELETE_WAIT:
			IF MC_BR_AsmDeleteShuttle_AcpTrak_0.Done THEN
				gTrakAsm.MonitorShuttlesPresent := 0;
				Step := COMMAND;
			END_IF

		//////////////////////////////////////////////////////////////////////////////////////////////////////////////////////////////
		// stop all shuttles in assembly
		STOP_SHUTTLE:
			CntShuttle := CntShuttle + 1;
			IF(CntShuttle > TRAK_MAX_SHUTTLE)THEN
				Step := READY;
			ELSIF(gTrakAsm.Shuttle[CntShuttle].Valid)THEN
				MC_Stop_0.Axis			:= ADR(gTrakAsm.Shuttle[CntShuttle].Axis);
				MC_Stop_0.Execute		:= TRUE;
				MC_Stop_0.Deceleration	:= gTrakAsm.ParaMoveDeceleration;
				MC_Stop_0.Jerk			:= 0.0;
				Step := STOP_SHUTTLE_WAIT;
			END_IF

		STOP_SHUTTLE_WAIT:
			Step := STOP_SHUTTLE;

		//////////////////////////////////////////////////////////////////////////////////////////////////////////////////////////////
		// move all shuttles

		// accelerate all shuttles in assembly via the same taget position to the same velocity
		// used for startup, to accelerate all shuttles to an initial velocity in order to pass the first process-point

		MOVE_SHUTTLE_VELOCITY:
			CntShuttle := CntShuttle + 1;
			IF(CntShuttle > TRAK_MAX_SHUTTLE)THEN
				Step := READY;
			ELSIF(gTrakAsm.Shuttle[CntShuttle].Valid)THEN
				MC_BR_RoutedMoveVel_AcpTrak_0.Axis			:= ADR(gTrakAsm.Shuttle[CntShuttle].Axis);
				MC_BR_RoutedMoveVel_AcpTrak_0.Execute		:= TRUE;
				MC_BR_RoutedMoveVel_AcpTrak_0.Sector		:= gTrakAsm.ParaMoveSectorRef;
				MC_BR_RoutedMoveVel_AcpTrak_0.Position		:= gTrakAsm.ParaMovePosition;
				MC_BR_RoutedMoveVel_AcpTrak_0.Velocity		:= gTrakAsm.ParaMoveVelocity;
				MC_BR_RoutedMoveVel_AcpTrak_0.RouteVelocity	:= gTrakAsm.ParaMoveRouteVelocity;
				MC_BR_RoutedMoveVel_AcpTrak_0.Acceleration	:= gTrakAsm.ParaMoveAcceleration;
				MC_BR_RoutedMoveVel_AcpTrak_0.Deceleration	:= gTrakAsm.ParaMoveDeceleration;
				MC_BR_RoutedMoveVel_AcpTrak_0.Jerk			:= 0.0;
				MC_BR_RoutedMoveVel_AcpTrak_0.BufferMode	:= mcABORTING;
				MC_BR_RoutedMoveVel_AcpTrak_0.AdvancedParameters.StartDirection		:= mcDIR_UNDEFINED;
				MC_BR_RoutedMoveVel_AcpTrak_0.AdvancedParameters.EndDirection		:= mcDIR_POSITIVE;
				MC_BR_RoutedMoveVel_AcpTrak_0.AdvancedParameters.ShuttleOrientation	:= mcDIR_UNDEFINED;
				Step := MOVE_SHUTTLE_VELOCITY_WAIT;
			END_IF

		MOVE_SHUTTLE_VELOCITY_WAIT:
			Step := MOVE_SHUTTLE_VELOCITY;

		// move all shuttles in assembly to the same target position
		// used to move all shuttles to a start position - one shuttle will reach this position, all the others are queuing up
		MOVE_SHUTTLE_POSITION:
			CntShuttle := CntShuttle + 1;
			IF(CntShuttle > TRAK_MAX_SHUTTLE)THEN
				Step := READY;
			ELSIF(gTrakAsm.Shuttle[CntShuttle].Valid)THEN
				MC_BR_RoutedMoveAbs_AcpTrak_0.Axis			:= ADR(gTrakAsm.Shuttle[CntShuttle].Axis);
				MC_BR_RoutedMoveAbs_AcpTrak_0.Execute		:= TRUE;
				MC_BR_RoutedMoveAbs_AcpTrak_0.Sector		:= gTrakAsm.ParaMoveSectorRef;
				MC_BR_RoutedMoveAbs_AcpTrak_0.Position		:= 0.0;//gTrakAsm.ParaMovePosition;
				MC_BR_RoutedMoveAbs_AcpTrak_0.Velocity		:= gTrakAsm.ParaMoveVelocity;
				MC_BR_RoutedMoveAbs_AcpTrak_0.Acceleration	:= gTrakAsm.ParaMoveAcceleration;
				MC_BR_RoutedMoveAbs_AcpTrak_0.Deceleration	:= gTrakAsm.ParaMoveDeceleration;
				MC_BR_RoutedMoveAbs_AcpTrak_0.Jerk			:= 0.0;
				MC_BR_RoutedMoveAbs_AcpTrak_0.BufferMode	:= mcABORTING;
				MC_BR_RoutedMoveAbs_AcpTrak_0.AdvancedParameters.StartDirection		:= mcDIR_UNDEFINED;
				MC_BR_RoutedMoveAbs_AcpTrak_0.AdvancedParameters.EndDirection		:= mcDIR_POSITIVE;
				MC_BR_RoutedMoveAbs_AcpTrak_0.AdvancedParameters.ShuttleOrientation	:= mcDIR_UNDEFINED;
				Step := MOVE_SHUTTLE_POSITION_WAIT;
			END_IF

		MOVE_SHUTTLE_POSITION_WAIT:
			Step := MOVE_SHUTTLE_POSITION;
	END_CASE

	//////////////////////////////////////////////////////////////////////////////////////////////////////////////////////////////
	// assembly FUBs

	MC_BR_AsmReset_AcpTrak_0.Assembly := gTrakAsm.AssemblyRef;
	MC_BR_AsmReset_AcpTrak_0();
	MC_BR_AsmReset_AcpTrak_0.Execute := FALSE;

	MC_BR_AsmPowerOn_AcpTrak_0.Assembly := gTrakAsm.AssemblyRef;
	MC_BR_AsmPowerOn_AcpTrak_0();
	MC_BR_AsmPowerOn_AcpTrak_0.Execute := FALSE;

	MC_BR_AsmPowerOff_AcpTrak_0.Assembly := gTrakAsm.AssemblyRef;
	MC_BR_AsmPowerOff_AcpTrak_0();
	MC_BR_AsmPowerOff_AcpTrak_0.Execute := FALSE;

	MC_BR_AsmGetInfo_AcpTrak_0.Assembly := gTrakAsm.AssemblyRef;
	MC_BR_AsmGetInfo_AcpTrak_0.Execute := TRUE;
	MC_BR_AsmGetInfo_AcpTrak_0();

	gTrakAsm.StatusSimulated := ((MC_BR_AsmGetInfo_AcpTrak_0.AssemblyInfo.SimulationOnPlcMode = mcACPTRAK_SIM_STATE_ON) OR DiagCpuIsSimulated() OR DiagCpuIsARsim());

	MC_BR_AsmReadStatus_AcpTrak_0.Assembly := gTrakAsm.AssemblyRef;
	MC_BR_AsmReadStatus_AcpTrak_0.Enable := TRUE;
	MC_BR_AsmReadStatus_AcpTrak_0();

	gTrakAsm.StatusDisabled		:= MC_BR_AsmReadStatus_AcpTrak_0.AssemblyDisabled;
	gTrakAsm.StatusReady		:= MC_BR_AsmReadStatus_AcpTrak_0.AssemblyReady;
	gTrakAsm.StatusHoming		:= MC_BR_AsmReadStatus_AcpTrak_0.AssemblyHoming;
	gTrakAsm.StatusStopping		:= MC_BR_AsmReadStatus_AcpTrak_0.AssemblyStopping;
	gTrakAsm.StatusErrorStop	:= MC_BR_AsmReadStatus_AcpTrak_0.AssemblyErrorStop;

	MC_BR_AsmReadInfo_AcpTrak_0.Assembly := gTrakAsm.AssemblyRef;
	MC_BR_AsmReadInfo_AcpTrak_0.Enable := TRUE;
	MC_BR_AsmReadInfo_AcpTrak_0();

	gTrakAsm.StatusCommunicationReady	:= MC_BR_AsmReadInfo_AcpTrak_0.AssemblyInfo.CommunicationReady;
	gTrakAsm.StatusReadyForPower		:= MC_BR_AsmReadInfo_AcpTrak_0.AssemblyInfo.ReadyForPowerOn;
	gTrakAsm.StatusPower				:= MC_BR_AsmReadInfo_AcpTrak_0.AssemblyInfo.PowerOn;
	gTrakAsm.MonitorShuttlesInErrorStop	:= MC_BR_AsmReadInfo_AcpTrak_0.AssemblyInfo.ShuttlesInErrorStopCount;
	gTrakAsm.MonitorSegmentsInErrorStop	:= MC_BR_AsmReadInfo_AcpTrak_0.AssemblyInfo.SegmentsInErrorStopCount;

	MC_BR_SecAddShuttle_AcpTrak_0();
	MC_BR_SecAddShuttle_AcpTrak_0.Execute := FALSE;

	MC_BR_AsmGetSegment_AcpTrak_0.Assembly := gTrakAsm.AssemblyRef;
	MC_BR_AsmGetSegment_AcpTrak_0();

	MC_BR_AsmGetShuttle_AcpTrak_0.Assembly := gTrakAsm.AssemblyRef;
	MC_BR_AsmGetShuttle_AcpTrak_0();

	MC_BR_AsmDeleteShuttle_AcpTrak_0.Assembly 	:= gTrakAsm.AssemblyRef;
	MC_BR_AsmDeleteShuttle_AcpTrak_0.Command	:= mcACPTRAK_SH_DELETE_ALL;
	MC_BR_AsmDeleteShuttle_AcpTrak_0();
	MC_BR_AsmDeleteShuttle_AcpTrak_0.Execute	:= FALSE;

	//////////////////////////////////////////////////////////////////////////////////////////////////////////////////////////////
	// segment FUBs

	FOR i:=1 TO TRAK_MAX_SEGMENT DO

		MC_BR_SegReadStatus_AcpTrak_0[i].Segment := ADR(gTrakAsm.Segment[i].Segment);
		MC_BR_SegReadStatus_AcpTrak_0[i].Enable  := (gTrakAsm.Segment[i].Segment.controlif <> 0);
		MC_BR_SegReadStatus_AcpTrak_0[i]();

		gTrakAsm.Segment[i].Valid := (MC_BR_SegReadStatus_AcpTrak_0[i].Valid);

		IF (gTrakAsm.Segment[i].Valid) THEN
			gTrakAsm.Segment[i].StatusDisabled 	:= MC_BR_SegReadStatus_AcpTrak_0[i].SegmentDisabled;
			gTrakAsm.Segment[i].StatusReady		:= MC_BR_SegReadStatus_AcpTrak_0[i].SegmentReady;
			gTrakAsm.Segment[i].StatusStopping	:= MC_BR_SegReadStatus_AcpTrak_0[i].SegmentStopping;
			gTrakAsm.Segment[i].StatusErrorStop	:= MC_BR_SegReadStatus_AcpTrak_0[i].SegmentErrorStop;
		END_IF

	END_FOR

	//////////////////////////////////////////////////////////////////////////////////////////////////////////////////////////////
	// shuttle FUBs

	FOR i:=1 TO TRAK_MAX_SHUTTLE DO

		MC_BR_ShReadInfo_AcpTrak_0[i].Axis		:= ADR(gTrakAsm.Shuttle[i].Axis);
		MC_BR_ShReadInfo_AcpTrak_0[i].Enable	:= (gTrakAsm.Shuttle[i].Axis.controlif <> 0);
		MC_BR_ShReadInfo_AcpTrak_0[i]();

		MC_ReadStatus_0[i].Axis		:= ADR(gTrakAsm.Shuttle[i].Axis);
		MC_ReadStatus_0[i].Enable	:= (gTrakAsm.Shuttle[i].Axis.controlif <> 0);
		MC_ReadStatus_0[i]();

		gTrakAsm.Shuttle[i].Valid := (MC_BR_ShReadInfo_AcpTrak_0[i].Valid AND MC_ReadStatus_0[i].Valid);
		IF(gTrakAsm.Shuttle[i].Valid)THEN
			gTrakAsm.Shuttle[i].ActSectorType		:= MC_BR_ShReadInfo_AcpTrak_0[i].ShuttleInfo.CurrentValues.SectorType;
			gTrakAsm.Shuttle[i].ActSector			:= MC_BR_ShReadInfo_AcpTrak_0[i].ShuttleInfo.CurrentValues.SectorName;
			gTrakAsm.Shuttle[i].ActPosition			:= MC_BR_ShReadInfo_AcpTrak_0[i].ShuttleInfo.CurrentValues.Position;
			gTrakAsm.Shuttle[i].ActVelocity			:= MC_BR_ShReadInfo_AcpTrak_0[i].ShuttleInfo.CurrentValues.Velocity;
			gTrakAsm.Shuttle[i].TotalMoveDistance	:= MC_BR_ShReadInfo_AcpTrak_0[i].ShuttleInfo.LifeCycleInfo.AbsoluteMovementDistance;
			gTrakAsm.Shuttle[i].StatusStandStill			:= MC_ReadStatus_0[i].StandStill;
			gTrakAsm.Shuttle[i].StatusStopping				:= MC_ReadStatus_0[i].Stopping;
			gTrakAsm.Shuttle[i].StatusErrorStop				:= MC_ReadStatus_0[i].ErrorStop;
			gTrakAsm.Shuttle[i].StatusDiscreteMotion		:= MC_ReadStatus_0[i].DiscreteMotion;
			gTrakAsm.Shuttle[i].StatusContinuousMotion		:= MC_ReadStatus_0[i].ContinuousMotion;
			gTrakAsm.Shuttle[i].StatusSynchronizedMotion	:= MC_ReadStatus_0[i].SynchronizedMotion;
		END_IF

	END_FOR

	MC_BR_ShCopyUserData_AcpTrak_0();
	MC_BR_ShCopyUserData_AcpTrak_0.Execute := FALSE;

	MC_Stop_0();
	MC_Stop_0.Execute := FALSE;

	MC_BR_RoutedMoveVel_AcpTrak_0();
	MC_BR_RoutedMoveVel_AcpTrak_0.Execute := FALSE;

	MC_BR_RoutedMoveAbs_AcpTrak_0();
	MC_BR_RoutedMoveAbs_AcpTrak_0.Execute := FALSE;

END_PROGRAM

PROGRAM _EXIT

END_PROGRAM
```

### Package Logical/Source/ProcessMachine - tasks to be used by the machine process

### gProcess.var
```iecst
(*Global Process Parameters*)
VAR
	gProductWidth : REAL := 0.15;
	gSpeedEmpty : REAL := 2.0;
	gAccEmpty : REAL := 20.0;
	gSpeedFull : REAL := 1.0;
	gAccFull : REAL := 10.0;
END_VAR
```

### Package Logical/Source/ProcessTemplate - template default tasks to be replicated

### Package Logical/Source/ProcessTemplate/SingleSh - single shuttle operation

### Program Logical/Source/ProcessTemplate/SingleSh/ProcInit (IEC) - trak process - init shuttles

#### Types.typ
```iecst
(*enum*)

TYPE
	StepEnum :
		(
		CHECK_TRIGGER := 0,
		GET_USERDATA,
		GET_USERDATA_WAIT,
		SET_USERDATA,
		SET_USERDATA_WAIT,
		GO_TO_NEXT_STATION
		);
END_TYPE
```

#### Main.st
```iecst
(*********************************************************************************
 * Copyright: 	B&R Industrial Automation GmbH
 * Author:    	B&R ES
 * Created:   	April 8, 2022/10:54 AM
 * Description:	All the shuttles crossing this process point will be considered
				initialized.
 * Mandatory: 	YES - Should be allways included in single shuttle station operations.
 *********************************************************************************)

PROGRAM _INIT

	(*******************************************************************)
	(******************* Process Configuration *************************)
	(*******************************************************************)
	PPAdr 	:= ADR(PP_Test); 	// <-- NAME A VALID PROCESS POINT
	(*** Define in/out speed & acceleration for this process ***)
	// OUT
	Speed_OUT ACCESS ADR(gSpeedEmpty); 	// <-- Bind it to Empty / Full speed global variable
	Acc_OUT	ACCESS ADR(gAccEmpty); 		// <-- Bind it to Empty / Full acceleration global variable
	(*** SceneViewer - Shuttle color after process ***)
	Red	  := 0.0;
	Green := 1.0;
	Blue  := 0.0;
	(********************************************************************)

	(* Local variable to enable/disable the process *)
	CmdEnableProcess := TRUE;
	(* Processpointreference for Functionblocks *)
	MC_BR_TrgPointEnable_AcpTrak_0.ProcessPoint 	:= PPAdr; // <-- NAME A VALID PROCESS POINT
	MC_BR_TrgPointGetInfo_AcpTrak_0.ProcessPoint 	:= PPAdr; // <-- NAME A VALID PROCESS POINT

END_PROGRAM

PROGRAM _CYCLIC

	//////////////////// HIGH PRIORITY ///////////////////
	IF gTrakAsm.StatusDisabled THEN
		Step 		:= CHECK_TRIGGER;
	END_IF
	//////////////////////////////////////////////////////

	CASE Step OF

		CHECK_TRIGGER:

			(* When the process is enabled and the assembly is ready, the process will be activated *)
			IF((CmdEnableProcess) AND (gTrakAsm.StatusReady))THEN
				MC_BR_TrgPointEnable_AcpTrak_0.Enable := TRUE;
				(* If a shuttle passes the triggerpoint then get the axis reference *)
				IF((MC_BR_TrgPointEnable_AcpTrak_0.Valid) AND (MC_BR_TrgPointEnable_AcpTrak_0.EventCount > 0))THEN
					MC_BR_TrgPointGetInfo_AcpTrak_0.Execute := TRUE;
				END_IF
			ELSE
				(* Else the processpoint will be disabled *)
				MC_BR_TrgPointEnable_AcpTrak_0.Enable := FALSE;
			END_IF

			(* If axis reference is available, save it and go to the next step *)
			IF EDGEPOS(MC_BR_TrgPointGetInfo_AcpTrak_0.Done) THEN
			(* Save axis reference in local variable for use in step machine *)
				ShuttleAxis	:= MC_BR_TrgPointGetInfo_AcpTrak_0.TrgPointInfo.Axis;
				Step 		:= GET_USERDATA;
			END_IF

		GET_USERDATA:

			(* The userdata is copied on a local variable *)
			MC_BR_ShCopyUserData_AcpTrak_0.Axis 		:= ADR(ShuttleAxis);
			MC_BR_ShCopyUserData_AcpTrak_0.Execute 		:= TRUE;
			MC_BR_ShCopyUserData_AcpTrak_0.DataAddress	:= ADR(ShuttleUserData);
			MC_BR_ShCopyUserData_AcpTrak_0.DataSize 	:= SIZEOF(ShuttleUserData);
			MC_BR_ShCopyUserData_AcpTrak_0.Mode 		:= mcACPTRAK_USERDATA_GET;

			Step := GET_USERDATA_WAIT;

		GET_USERDATA_WAIT:

			(* After copying go to the next step *)
			IF (MC_BR_ShCopyUserData_AcpTrak_0.Done) THEN
				IF ShuttleUserData.InitDone THEN
					Step := CHECK_TRIGGER;
				ELSE
					Step := SET_USERDATA;
				END_IF
			END_IF

		SET_USERDATA:

			(* Change color to know that shuttles are in unsync. *)
			ShuttleUserData.SceneColorRed 	:= Red;
			ShuttleUserData.SceneColorGreen := Green;
			ShuttleUserData.SceneColorBlue	:= Blue;

			(* After this point, the shuttle is initialized *)
			ShuttleUserData.InitDone := TRUE;

			(* The modified userdata will be copied back on the shuttle *)
			MC_BR_ShCopyUserData_AcpTrak_0.Axis 		:= ADR(ShuttleAxis);
			MC_BR_ShCopyUserData_AcpTrak_0.Execute 		:= TRUE;
			MC_BR_ShCopyUserData_AcpTrak_0.DataAddress	:= ADR(ShuttleUserData);
			MC_BR_ShCopyUserData_AcpTrak_0.DataSize 	:= SIZEOF(ShuttleUserData);
			MC_BR_ShCopyUserData_AcpTrak_0.Mode 		:= mcACPTRAK_USERDATA_SET;
			Step := SET_USERDATA_WAIT;

		SET_USERDATA_WAIT:

			IF (MC_BR_ShCopyUserData_AcpTrak_0.Done) THEN
				Step := GO_TO_NEXT_STATION;
			END_IF

		GO_TO_NEXT_STATION:

			MC_BR_ElasticMoveVel_AcpTrak_0.Axis 	:= ADR(ShuttleAxis);
			MC_BR_ElasticMoveVel_AcpTrak_0.Execute	:= TRUE;

			Step := CHECK_TRIGGER;

	END_CASE

	(*** Call all function blocks ***)
	// MC_BR_TrgPointEnable_AcpTrak
	MC_BR_TrgPointEnable_AcpTrak_0();
	// MC_BR_TrgPointGetInfo_AcpTrak
	MC_BR_TrgPointGetInfo_AcpTrak_0();
	MC_BR_TrgPointGetInfo_AcpTrak_0.Execute  := FALSE;
	// MC_BR_ShCopyUserData_AcpTrak
	MC_BR_ShCopyUserData_AcpTrak_0();
	MC_BR_ShCopyUserData_AcpTrak_0.Execute 	 := FALSE;
	//MC_BR_ElasticMoveVel_AcpTrak_0
	MC_BR_ElasticMoveVel_AcpTrak_0.Velocity		:= Speed_OUT;
	MC_BR_ElasticMoveVel_AcpTrak_0.Acceleration	:= Acc_OUT;
	MC_BR_ElasticMoveVel_AcpTrak_0.Deceleration	:= Acc_OUT;
	MC_BR_ElasticMoveVel_AcpTrak_0.Direction	:= mcDIR_POSITIVE;
	MC_BR_ElasticMoveVel_AcpTrak_0();
	MC_BR_ElasticMoveVel_AcpTrak_0.Execute		:= FALSE;

END_PROGRAM
```

### Program Logical/Source/ProcessTemplate/SingleSh/ProcStop_S1 (IEC) - trak process - 1 shuttle wait predefined time

#### Types.typ
```iecst
(*enum*)

TYPE
	StepEnum :
		(
		CHECK_TRIGGER,
		GET_SHUTTLE_DATA,
		GET_SHUTTLE_DATA_WAIT,
		GO_TO_PROCESS_STATION,
		GO_TO_PROCESS_STATION_WAIT,
		WAIT,
		SET_SHUTTLE_DATA,
		SET_SHUTTLE_DATA_WAIT,
		GO_TO_NEXT_STATION
		);
	StepTicket :
		(
		ENABLE_BARRIER := 0,
		OPENED_BARRIER,
		FREE_SHUTTLES
		);
END_TYPE
```

#### Variables.var
```iecst
(*process configuration*)
VAR
	PPAdr : UDINT;
	SecAdr : UDINT;
END_VAR
(*commands*)
VAR
	CmdEnableProcess : BOOL;
END_VAR
(*sequence control*)
VAR
	Step : StepEnum;
	ShuttleAxis : McAxisType;
	ShuttleUserData : TrakShuttleUserDataType;
	WaitTime : UDINT := 500;
	ProcPointPos : LREAL;
	DistTravelled : LREAL;
	ReleaseSts : BOOL;
END_VAR
(*barrier functionality*)
VAR
	sTickets : StepTicket; (*step variable for state machine*)
	cmdFreeShuttles : BOOL; (*When should the shuttles be released*)
END_VAR
(*colour configuration*)
VAR
	Red : REAL;
	Green : REAL;
	Blue : REAL;
END_VAR
(*movement configuration*)
VAR
	Speed_IN : REFERENCE TO REAL;
	Acc_IN : REFERENCE TO REAL;
	Speed_OUT : REFERENCE TO REAL;
	Acc_OUT : REFERENCE TO REAL;
END_VAR
(*FUB - Generic*)
VAR
	MC_BR_AsmReadStatus_AcpTrak_0 : MC_BR_AsmReadStatus_AcpTrak;
	MC_BR_TrgPointEnable_AcpTrak_0 : MC_BR_TrgPointEnable_AcpTrak;
	MC_BR_TrgPointGetInfo_AcpTrak_0 : MC_BR_TrgPointGetInfo_AcpTrak;
	MC_BR_ShCopyUserData_AcpTrak_0 : MC_BR_ShCopyUserData_AcpTrak;
	MC_BR_RoutedMoveAbs_AcpTrak_0 : MC_BR_RoutedMoveAbs_AcpTrak;
	MC_BR_ElasticMoveVel_AcpTrak_0 : MC_BR_ElasticMoveVel_AcpTrak;
	MC_BR_ProcPointGetInfo_AcpTrak_0 : MC_BR_ProcPointGetInfo_AcpTrak;
	TON_0 : TON;
END_VAR
(*FUB - Barrier*)
VAR
	MC_BR_BarrierCommand_AcpTrak_0 : MC_BR_BarrierCommand_AcpTrak;
	MC_BR_BarrierReadInfo_AcpTrak_0 : MC_BR_BarrierReadInfo_AcpTrak;
END_VAR
```

#### Main.st
```iecst
(*********************************************************************************
 * Copyright: 	B&R Industrial Automation GmbH
 * Author:    	B&R ES
 * Created:   	April 8, 2022/10:54 AM
 * Description:	A single shuttle will be stopped a predefined time in the process
				station.
 * Mandatory: 	NO
 *********************************************************************************)
PROGRAM _INIT

	(*******************************************************************)
	(******************* Process Configuration *************************)
	(*******************************************************************)
	PPAdr 	:= ADR(PP_Test); 		// <-- NAME A VALID PROCESS POINT
	SecAdr	:= ADR(SectorTrackA);	// <-- NAME A VALID SECTOR
	(*** Define in/out speed & acceleration for this process ***)
	// IN
	Speed_IN ACCESS	ADR(gSpeedEmpty); 	// <-- Bind it to Empty / Full speed global variable
	Acc_IN ACCESS ADR(gAccEmpty); 		// <-- Bind it to Empty / Full acceleration global variable
	// OUT
	Speed_OUT ACCESS ADR(gSpeedFull); 	// <-- Bind it to Empty / Full speed global variable
	Acc_OUT	ACCESS ADR(gAccFull); 		// <-- Bind it to Empty / Full acceleration global variable
	(*** Define Wait Time (ms) ***)
	WaitTime := 500;
	(*** Define stop distance for the shuttles ***)
	DistTravelled	:= 0.33;
	(*** Define if it is a release station ***)
	ReleaseSts := FALSE;
	(*** SceneViewer - Shuttle color after process ***)
	Red	  := 0.02;
	Green := 0.77;
	Blue  := 0.21;
	(********************************************************************)

	CmdEnableProcess 	:= TRUE;
	cmdFreeShuttles		:= TRUE;
	Step 				:= CHECK_TRIGGER;

	MC_BR_ProcPointGetInfo_AcpTrak_0.ProcessPoint   := PPAdr;
	MC_BR_ProcPointGetInfo_AcpTrak_0.Execute		:= TRUE;

	REPEAT
		MC_BR_ProcPointGetInfo_AcpTrak_0();
	UNTIL
		MC_BR_ProcPointGetInfo_AcpTrak_0.Done OR MC_BR_ProcPointGetInfo_AcpTrak_0.Error
	END_REPEAT;

	ProcPointPos 	:= MC_BR_ProcPointGetInfo_AcpTrak_0.ProcPointInfo.SectorPosition.Position;

END_PROGRAM

PROGRAM _CYCLIC

	///////////////// HIGH PRIORITY /////////////////
	(* reset process sequence if assembly is disabled *)
	IF EDGEPOS(gTrakAsm.StatusDisabled) THEN
		TON_0.IN		:= FALSE;
		cmdFreeShuttles	:= (MC_BR_BarrierReadInfo_AcpTrak_0.BarrierInfo.RemainingTickets = 0);
		Step 			:= CHECK_TRIGGER;
	END_IF

	///////////// BARRIER FUNCTIONALITY /////////////
	(* this state machine is developed in such a way that allows to enable/disable the station without having to stop *)
	CASE sTickets OF
		ENABLE_BARRIER:
			MC_BR_BarrierCommand_AcpTrak_0.ProcessPoint := PPAdr;
			IF CmdEnableProcess THEN
				MC_BR_BarrierCommand_AcpTrak_0.Command := mcACPTRAK_BARRIER_CLOSE;
			ELSE
				MC_BR_BarrierCommand_AcpTrak_0.Command := mcACPTRAK_BARRIER_OPEN;
			END_IF
			MC_BR_BarrierCommand_AcpTrak_0.Execute := TRUE;
			IF (MC_BR_BarrierCommand_AcpTrak_0.Done) THEN
				MC_BR_BarrierCommand_AcpTrak_0.Execute := FALSE;
				IF CmdEnableProcess THEN
					sTickets := FREE_SHUTTLES;
				ELSE
					sTickets := OPENED_BARRIER;
				END_IF
			END_IF
		OPENED_BARRIER:
			IF EDGEPOS(CmdEnableProcess) THEN
				cmdFreeShuttles := (MC_BR_BarrierReadInfo_AcpTrak_0.BarrierInfo.RemainingTickets = 0);
				sTickets 		:= ENABLE_BARRIER;
			END_IF
		FREE_SHUTTLES:
			IF cmdFreeShuttles THEN
				MC_BR_BarrierCommand_AcpTrak_0.Command 							:= mcACPTRAK_BARRIER_ADD_TICKETS;
				MC_BR_BarrierCommand_AcpTrak_0.AdvancedParameters.TicketCount 	:= 1;
				MC_BR_BarrierCommand_AcpTrak_0.Execute 							:= TRUE;
				IF (MC_BR_BarrierCommand_AcpTrak_0.Done) THEN
					MC_BR_BarrierCommand_AcpTrak_0.Execute := FALSE;
					cmdFreeShuttles := FALSE;
				END_IF
			END_IF
			IF EDGENEG(CmdEnableProcess) THEN
				sTickets := ENABLE_BARRIER;
			END_IF
	END_CASE

	(***********************************************************************)
	(************************* STATE MACHINE *******************************)
	(***********************************************************************)

	CASE Step OF

		(* enable trigger and wait for one shuttle to pass *)
		CHECK_TRIGGER:
			IF((CmdEnableProcess) AND (MC_BR_AsmReadStatus_AcpTrak_0.AssemblyReady))THEN
				MC_BR_TrgPointEnable_AcpTrak_0.ProcessPoint  := PPAdr;
				MC_BR_TrgPointEnable_AcpTrak_0.Enable        := TRUE;
				(* shuttle passed => get axis reference *)
				IF((MC_BR_TrgPointEnable_AcpTrak_0.Valid) AND (MC_BR_TrgPointEnable_AcpTrak_0.EventCount > 0))THEN
					MC_BR_TrgPointGetInfo_AcpTrak_0.ProcessPoint  := PPAdr;
					MC_BR_TrgPointGetInfo_AcpTrak_0.Execute       := TRUE;
					Step := GET_SHUTTLE_DATA;
				END_IF
			ELSE
				MC_BR_TrgPointEnable_AcpTrak_0.Enable  := FALSE;
			END_IF

			(* axis reference of passed shuttle available *)
			(* get shuttle-UserData *)
		GET_SHUTTLE_DATA:

			IF(MC_BR_TrgPointGetInfo_AcpTrak_0.Done)THEN
				ShuttleAxis := MC_BR_TrgPointGetInfo_AcpTrak_0.TrgPointInfo.Axis;
				// read UserData from shuttle
				MC_BR_ShCopyUserData_AcpTrak_0.Axis         := ADR(ShuttleAxis);
				MC_BR_ShCopyUserData_AcpTrak_0.Execute      := TRUE;
				MC_BR_ShCopyUserData_AcpTrak_0.DataAddress  := ADR(ShuttleUserData);
				MC_BR_ShCopyUserData_AcpTrak_0.DataSize     := SIZEOF(ShuttleUserData);
				MC_BR_ShCopyUserData_AcpTrak_0.Mode         := mcACPTRAK_USERDATA_GET;
				Step := GET_SHUTTLE_DATA_WAIT;
			END_IF

			(* wait for shuttle-UserData content available *)
		GET_SHUTTLE_DATA_WAIT:
			IF(MC_BR_ShCopyUserData_AcpTrak_0.Done)THEN
				IF ShuttleUserData.InitDone THEN
					Step 			:= GO_TO_PROCESS_STATION;
				ELSE
					cmdFreeShuttles := (MC_BR_BarrierReadInfo_AcpTrak_0.BarrierInfo.RemainingTickets = 0);
					Step 			:= CHECK_TRIGGER;
				END_IF
			END_IF

		GO_TO_PROCESS_STATION:

			MC_BR_RoutedMoveAbs_AcpTrak_0.Axis		:= ADR(ShuttleAxis);
			MC_BR_RoutedMoveAbs_AcpTrak_0.Position 	:= ProcPointPos + DistTravelled;
			MC_BR_RoutedMoveAbs_AcpTrak_0.Execute 	:= TRUE;

			Step 		:= GO_TO_PROCESS_STATION_WAIT;

		GO_TO_PROCESS_STATION_WAIT:

			IF (MC_BR_RoutedMoveAbs_AcpTrak_0.Done) THEN
				TON_0.IN 	:= TRUE;
				Step 		:= WAIT;
			END_IF

		WAIT:

			IF TON_0.Q THEN
				TON_0.IN 	:= FALSE;
				Step 		:= SET_SHUTTLE_DATA;
			END_IF

		(* write modified UserData back to shuttle *)
		SET_SHUTTLE_DATA:

			ShuttleUserData.SceneColorRed	:= Red;
			ShuttleUserData.SceneColorGreen	:= Green;
			ShuttleUserData.SceneColorBlue 	:= Blue;

			MC_BR_ShCopyUserData_AcpTrak_0.Axis         := ADR(ShuttleAxis);
			MC_BR_ShCopyUserData_AcpTrak_0.Execute      := TRUE;
			MC_BR_ShCopyUserData_AcpTrak_0.DataAddress  := ADR(ShuttleUserData);
			MC_BR_ShCopyUserData_AcpTrak_0.DataSize     := SIZEOF(ShuttleUserData);
			MC_BR_ShCopyUserData_AcpTrak_0.Mode         := mcACPTRAK_USERDATA_SET;
			Step := SET_SHUTTLE_DATA_WAIT;

		(* wait for shuttle-UserData content set *)
		SET_SHUTTLE_DATA_WAIT:

			IF(MC_BR_ShCopyUserData_AcpTrak_0.Done)THEN
				Step	 	:= GO_TO_NEXT_STATION;
			END_IF

		(* go to next station *)
		GO_TO_NEXT_STATION:

			MC_BR_ElasticMoveVel_AcpTrak_0.Axis           := ADR(ShuttleAxis);
			MC_BR_ElasticMoveVel_AcpTrak_0.Execute        := TRUE;

			IF ReleaseSts THEN
				gProducedProduct := gProducedProduct + 1;
			END_IF

			cmdFreeShuttles := TRUE;
			Step 			:= CHECK_TRIGGER;

	END_CASE

	(*** Call all function blocks ***)
	// MC_BR_AsmReadStatus_AcpTrak
	MC_BR_AsmReadStatus_AcpTrak_0.Assembly 	:= ADR(gAssembly_1);
	MC_BR_AsmReadStatus_AcpTrak_0.Enable 	:= TRUE;
	MC_BR_AsmReadStatus_AcpTrak_0();
    // MC_BR_TrgPointEnable_AcpTrak
	MC_BR_TrgPointEnable_AcpTrak_0();
    // MC_BR_TrgPointGetInfo_AcpTrak
	MC_BR_TrgPointGetInfo_AcpTrak_0();
	MC_BR_TrgPointGetInfo_AcpTrak_0.Execute := FALSE;
    // TON_0
	TON_0.PT := UDINT_TO_TIME(WaitTime);
	TON_0();
	// MC_BR_ShCopyUserData_AcpTrak
	MC_BR_ShCopyUserData_AcpTrak_0();
	MC_BR_ShCopyUserData_AcpTrak_0.Execute := FALSE;
	// MC_BR_RoutedMoveAbs_AcpTrak_0
	MC_BR_RoutedMoveAbs_AcpTrak_0.Sector 		  := SecAdr;
	MC_BR_RoutedMoveAbs_AcpTrak_0.Velocity		  := Speed_IN;
	MC_BR_RoutedMoveAbs_AcpTrak_0.Acceleration	  := Acc_IN;
	MC_BR_RoutedMoveAbs_AcpTrak_0.Deceleration	  := Acc_IN;
	MC_BR_RoutedMoveAbs_AcpTrak_0();
	MC_BR_RoutedMoveAbs_AcpTrak_0.Execute := FALSE;
	// MC_BR_ElasticMoveVel_AcpTrak_0
	MC_BR_ElasticMoveVel_AcpTrak_0.Velocity       := Speed_OUT;
	MC_BR_ElasticMoveVel_AcpTrak_0.Acceleration   := Acc_OUT;
	MC_BR_ElasticMoveVel_AcpTrak_0.Deceleration   := Acc_OUT;
	MC_BR_ElasticMoveVel_AcpTrak_0.Jerk           := 0.0;
	MC_BR_ElasticMoveVel_AcpTrak_0.Direction	  := mcDIR_POSITIVE;
	MC_BR_ElasticMoveVel_AcpTrak_0.BufferMode     := mcABORTING;
	MC_BR_ElasticMoveVel_AcpTrak_0();
	MC_BR_ElasticMoveVel_AcpTrak_0.Execute := FALSE;
	//MC_BR_BarrierCommand_AcpTrak
	MC_BR_BarrierCommand_AcpTrak_0();
	//MC_BR_BarrierReadInfo_AcpTrak
	MC_BR_BarrierReadInfo_AcpTrak_0.ProcessPoint := PPAdr;
	MC_BR_BarrierReadInfo_AcpTrak_0.Enable		 := TRUE;
	MC_BR_BarrierReadInfo_AcpTrak_0();

END_PROGRAM
```

### Program Logical/Source/ProcessTemplate/SingleSh/ProcStop_S2 (IEC) - trak process - 2 shuttles wait predefined time

#### Types.typ
```iecst
(*enum*)

TYPE
	StepEnum :
		(
		CHECK_TRIGGER,
		GET_SHUTTLE_DATA,
		GET_SHUTTLE_DATA_WAIT,
		GO_TO_PROCESS_STATION_1,
		GO_TO_PROCESS_STATION_2,
		GO_TO_PROCESS_STATION_WAIT,
		WAIT,
		SET_SHUTTLE_DATA,
		SET_SHUTTLE_DATA_WAIT,
		GO_TO_NEXT_STATION
		);
	StepTicket :
		(
		ENABLE_BARRIER := 0,
		OPENED_BARRIER,
		FREE_SHUTTLES
		);
END_TYPE
```

#### Variables.var
```iecst
(*process configuration*)
VAR
	PPAdr : UDINT;
	SecAdr : UDINT;
END_VAR
(*commands*)
VAR
	CmdEnableProcess : BOOL;
END_VAR
(*sequence control*)
VAR
	Step : StepEnum;
	ShuttleAxis : ARRAY[1..2] OF McAxisType;
	ShuttleUserData : ARRAY[1..2] OF TrakShuttleUserDataType;
	WaitTime : UDINT := 500;
	ProcPointPos : LREAL;
	CntShuttle : USINT;
	DistTravelled_1 : LREAL;
	DistTravelled_2 : LREAL;
	ReleaseSts : BOOL;
END_VAR
(*barrier functionality*)
VAR
	sTickets : StepTicket; (*step variable for state machine*)
	cmdFreeShuttles : BOOL; (*When should the shuttles be released*)
END_VAR
(*colour configuration*)
VAR
	Red : REAL;
	Green : REAL;
	Blue : REAL;
END_VAR
(*movement configuration*)
VAR
	Speed_IN : REFERENCE TO REAL;
	Acc_IN : REFERENCE TO REAL;
	Speed_OUT : REFERENCE TO REAL;
	Acc_OUT : REFERENCE TO REAL;
END_VAR
(*FUB - Generic*)
VAR
	MC_BR_AsmReadStatus_AcpTrak_0 : MC_BR_AsmReadStatus_AcpTrak;
	MC_BR_TrgPointEnable_AcpTrak_0 : MC_BR_TrgPointEnable_AcpTrak;
	MC_BR_TrgPointGetInfo_AcpTrak_0 : MC_BR_TrgPointGetInfo_AcpTrak;
	MC_BR_ShCopyUserData_AcpTrak_0 : MC_BR_ShCopyUserData_AcpTrak;
	MC_BR_RoutedMoveAbs_AcpTrak_0 : MC_BR_RoutedMoveAbs_AcpTrak;
	MC_BR_ElasticMoveVel_AcpTrak_0 : MC_BR_ElasticMoveVel_AcpTrak;
	MC_BR_ProcPointGetInfo_AcpTrak_0 : MC_BR_ProcPointGetInfo_AcpTrak;
	MC_ReadStatus_0 : MC_ReadStatus;
	MC_ReadStatus_1 : MC_ReadStatus;
	TON_0 : TON;
END_VAR
(*FUB - Barrier*)
VAR
	MC_BR_BarrierCommand_AcpTrak_0 : MC_BR_BarrierCommand_AcpTrak;
	MC_BR_BarrierReadInfo_AcpTrak_0 : MC_BR_BarrierReadInfo_AcpTrak;
END_VAR
```

#### Main.st
```iecst
(*********************************************************************************
 * Copyright: 	B&R Industrial Automation GmbH
 * Author:    	B&R ES
 * Created:   	April 8, 2022/10:54 AM
 * Description:	Two shuttles will be stopped a predefined time in the process
				station.
 * Mandatory: 	NO
 *********************************************************************************)
PROGRAM _INIT

	(*******************************************************************)
	(******************* Process Configuration *************************)
	(*******************************************************************)
	PPAdr 	:= ADR(PP_Test); 		// <-- NAME A VALID PROCESS POINT
	SecAdr	:= ADR(SectorTrackA);	// <-- NAME A VALID SECTOR
	(*** Define in/out speed & acceleration for this process ***)
	// IN
	Speed_IN ACCESS	ADR(gSpeedEmpty); 	// <-- Bind it to Empty / Full speed global variable
	Acc_IN ACCESS ADR(gAccEmpty); 		// <-- Bind it to Empty / Full acceleration global variable
	// OUT
	Speed_OUT ACCESS ADR(gSpeedFull); 	// <-- Bind it to Empty / Full speed global variable
	Acc_OUT	ACCESS ADR(gAccFull); 		// <-- Bind it to Empty / Full acceleration global variable
	(*** Define Wait Time (ms) ***)
	WaitTime := 500;
	(*** Define relative center point distance for the first coupled shuttles ***)
	DistTravelled_1	:= 0.66;
	DistTravelled_2 := 0.33;
	(*** Define if it is a release station ***)
	ReleaseSts := FALSE;
	(*** SceneViewer - Shuttle color after process ***)
	Red	  := 0.02;
	Green := 0.77;
	Blue  := 0.21;
	(********************************************************************)

	CmdEnableProcess 	:= TRUE;
	cmdFreeShuttles		:= TRUE;
	Step 				:= CHECK_TRIGGER;

	MC_BR_ProcPointGetInfo_AcpTrak_0.ProcessPoint   := PPAdr;
	MC_BR_ProcPointGetInfo_AcpTrak_0.Execute		:= TRUE;

	REPEAT
		MC_BR_ProcPointGetInfo_AcpTrak_0();
	UNTIL
		MC_BR_ProcPointGetInfo_AcpTrak_0.Done OR MC_BR_ProcPointGetInfo_AcpTrak_0.Error
	END_REPEAT;

	ProcPointPos 	:= MC_BR_ProcPointGetInfo_AcpTrak_0.ProcPointInfo.SectorPosition.Position;
	CntShuttle 		:= 1;

END_PROGRAM

PROGRAM _CYCLIC

	///////////////// HIGH PRIORITY /////////////////
	(* reset process sequence if assembly is disabled *)
	IF EDGEPOS(gTrakAsm.StatusDisabled) THEN
		CntShuttle 		:= 1;
		TON_0.IN		:= FALSE;
		cmdFreeShuttles	:= (MC_BR_BarrierReadInfo_AcpTrak_0.BarrierInfo.RemainingTickets = 0);
		Step 			:= CHECK_TRIGGER;
	END_IF

	///////////// BARRIER FUNCTIONALITY /////////////
	(* this state machine is developed in such a way that allows to enable/disable the station without having to stop *)
	CASE sTickets OF
		ENABLE_BARRIER:
			MC_BR_BarrierCommand_AcpTrak_0.ProcessPoint := PPAdr;
			IF CmdEnableProcess THEN
				MC_BR_BarrierCommand_AcpTrak_0.Command := mcACPTRAK_BARRIER_CLOSE;
			ELSE
				MC_BR_BarrierCommand_AcpTrak_0.Command := mcACPTRAK_BARRIER_OPEN;
			END_IF
			MC_BR_BarrierCommand_AcpTrak_0.Execute := TRUE;
			IF (MC_BR_BarrierCommand_AcpTrak_0.Done) THEN
				MC_BR_BarrierCommand_AcpTrak_0.Execute := FALSE;
				IF CmdEnableProcess THEN
					sTickets := FREE_SHUTTLES;
				ELSE
					sTickets := OPENED_BARRIER;
				END_IF
			END_IF
		OPENED_BARRIER:
			IF EDGEPOS(CmdEnableProcess) THEN
				cmdFreeShuttles := (MC_BR_BarrierReadInfo_AcpTrak_0.BarrierInfo.RemainingTickets = 0);
				sTickets 		:= ENABLE_BARRIER;
			END_IF
		FREE_SHUTTLES:
			IF cmdFreeShuttles THEN
				MC_BR_BarrierCommand_AcpTrak_0.Command 							:= mcACPTRAK_BARRIER_ADD_TICKETS;
				MC_BR_BarrierCommand_AcpTrak_0.AdvancedParameters.TicketCount 	:= 1;
				MC_BR_BarrierCommand_AcpTrak_0.Execute 							:= TRUE;
				IF (MC_BR_BarrierCommand_AcpTrak_0.Done) THEN
					MC_BR_BarrierCommand_AcpTrak_0.Execute := FALSE;
					cmdFreeShuttles := FALSE;
				END_IF
			END_IF
			IF EDGENEG(CmdEnableProcess) THEN
				sTickets := ENABLE_BARRIER;
			END_IF
	END_CASE

	(***********************************************************************)
	(************************* STATE MACHINE *******************************)
	(***********************************************************************)

	CASE Step OF

		(* enable trigger and wait for one shuttle to pass *)
		CHECK_TRIGGER:
			IF((CmdEnableProcess) AND (MC_BR_AsmReadStatus_AcpTrak_0.AssemblyReady))THEN
				MC_BR_TrgPointEnable_AcpTrak_0.ProcessPoint  := PPAdr;
				MC_BR_TrgPointEnable_AcpTrak_0.Enable        := TRUE;
				(* shuttle passed => get axis reference *)
				IF((MC_BR_TrgPointEnable_AcpTrak_0.Valid) AND (MC_BR_TrgPointEnable_AcpTrak_0.EventCount > 0))THEN
					MC_BR_TrgPointGetInfo_AcpTrak_0.ProcessPoint  := PPAdr;
					MC_BR_TrgPointGetInfo_AcpTrak_0.Execute       := TRUE;
					Step := GET_SHUTTLE_DATA;
				END_IF
			ELSE
				MC_BR_TrgPointEnable_AcpTrak_0.Enable  := FALSE;
			END_IF

		(* axis reference of passed shuttle available *)
		(* get shuttle-UserData *)
		GET_SHUTTLE_DATA:

			IF(MC_BR_TrgPointGetInfo_AcpTrak_0.Done)THEN
				ShuttleAxis[CntShuttle] := MC_BR_TrgPointGetInfo_AcpTrak_0.TrgPointInfo.Axis;
				// read UserData from shuttle
				MC_BR_ShCopyUserData_AcpTrak_0.Axis         := ADR(ShuttleAxis[CntShuttle]);
				MC_BR_ShCopyUserData_AcpTrak_0.Execute      := TRUE;
				MC_BR_ShCopyUserData_AcpTrak_0.DataAddress  := ADR(ShuttleUserData[CntShuttle]);
				MC_BR_ShCopyUserData_AcpTrak_0.DataSize     := SIZEOF(ShuttleUserData[CntShuttle]);
				MC_BR_ShCopyUserData_AcpTrak_0.Mode         := mcACPTRAK_USERDATA_GET;
				Step := GET_SHUTTLE_DATA_WAIT;
			END_IF

		(* wait for shuttle-UserData content available *)
		GET_SHUTTLE_DATA_WAIT:
			IF(MC_BR_ShCopyUserData_AcpTrak_0.Done)THEN
				IF ShuttleUserData[CntShuttle].InitDone THEN
					CASE CntShuttle OF
						//First shuttle
						1:
							Step := GO_TO_PROCESS_STATION_1;
						// Second shuttle
						2:
							Step := GO_TO_PROCESS_STATION_2;
					END_CASE
				ELSE
					cmdFreeShuttles := (MC_BR_BarrierReadInfo_AcpTrak_0.BarrierInfo.RemainingTickets = 0);
					Step 			:= CHECK_TRIGGER;
				END_IF
			END_IF

		GO_TO_PROCESS_STATION_1:

			MC_BR_RoutedMoveAbs_AcpTrak_0.Axis			:= ADR(ShuttleAxis[CntShuttle]);
			MC_BR_RoutedMoveAbs_AcpTrak_0.Position 		:= ProcPointPos + DistTravelled_1;
			MC_BR_RoutedMoveAbs_AcpTrak_0.Execute 		:= TRUE;

			CntShuttle 		:= CntShuttle + 1;
			cmdFreeShuttles := TRUE;
			Step 			:= CHECK_TRIGGER;

		GO_TO_PROCESS_STATION_2:

			MC_BR_RoutedMoveAbs_AcpTrak_0.Axis			:= ADR(ShuttleAxis[CntShuttle]);
			MC_BR_RoutedMoveAbs_AcpTrak_0.Position 		:= ProcPointPos + DistTravelled_2;
			MC_BR_RoutedMoveAbs_AcpTrak_0.Execute 		:= TRUE;

			Step 		:= GO_TO_PROCESS_STATION_WAIT;

		GO_TO_PROCESS_STATION_WAIT:

			MC_ReadStatus_0.Axis 	:= ADR(ShuttleAxis[1]);
			MC_ReadStatus_0.Enable	:= TRUE;

			MC_ReadStatus_1.Axis 	:= ADR(ShuttleAxis[2]);
			MC_ReadStatus_1.Enable	:= TRUE;

			IF (MC_ReadStatus_0.StandStill AND MC_ReadStatus_1.StandStill) THEN
				MC_ReadStatus_0.Enable := FALSE;
				MC_ReadStatus_1.Enable := FALSE;
				TON_0.IN 	:= TRUE;
				Step 		:= WAIT;
			END_IF

		WAIT:

			IF TON_0.Q THEN
				TON_0.IN 	:= FALSE;
				CntShuttle 	:= 1;
				Step 		:= SET_SHUTTLE_DATA;
			END_IF

		(* write modified UserData back to shuttle *)
		SET_SHUTTLE_DATA:

			ShuttleUserData[CntShuttle].SceneColorRed	:= Red;
			ShuttleUserData[CntShuttle].SceneColorGreen	:= Green;
			ShuttleUserData[CntShuttle].SceneColorBlue 	:= Blue;

			MC_BR_ShCopyUserData_AcpTrak_0.Axis         := ADR(ShuttleAxis[CntShuttle]);
			MC_BR_ShCopyUserData_AcpTrak_0.Execute      := TRUE;
			MC_BR_ShCopyUserData_AcpTrak_0.DataAddress  := ADR(ShuttleUserData[CntShuttle]);
			MC_BR_ShCopyUserData_AcpTrak_0.DataSize     := SIZEOF(ShuttleUserData[CntShuttle]);
			MC_BR_ShCopyUserData_AcpTrak_0.Mode         := mcACPTRAK_USERDATA_SET;
			Step := SET_SHUTTLE_DATA_WAIT;

		(* wait for shuttle-UserData content set *)
		SET_SHUTTLE_DATA_WAIT:

			IF(MC_BR_ShCopyUserData_AcpTrak_0.Done)THEN
				Step := GO_TO_NEXT_STATION;
			END_IF

			(* go to next station *)
		GO_TO_NEXT_STATION:

			MC_BR_ElasticMoveVel_AcpTrak_0.Axis           := ADR(ShuttleAxis[CntShuttle]);
			MC_BR_ElasticMoveVel_AcpTrak_0.Execute        := TRUE;

			IF ReleaseSts THEN
				gProducedProduct := gProducedProduct + 2;
			END_IF

			CASE CntShuttle OF
				1:
					CntShuttle 	:= CntShuttle + 1;
					Step		:= SET_SHUTTLE_DATA;
				2:
					CntShuttle		:= 1;
					cmdFreeShuttles	:= TRUE;
					Step 			:= CHECK_TRIGGER;
			END_CASE

	END_CASE

	(*** Call all function blocks ***)
	// MC_BR_AsmReadStatus_AcpTrak
	MC_BR_AsmReadStatus_AcpTrak_0.Assembly 	:= ADR(gAssembly_1);
	MC_BR_AsmReadStatus_AcpTrak_0.Enable 	:= TRUE;
	MC_BR_AsmReadStatus_AcpTrak_0();
    // MC_BR_TrgPointEnable_AcpTrak
	MC_BR_TrgPointEnable_AcpTrak_0();
    // MC_BR_TrgPointGetInfo_AcpTrak
	MC_BR_TrgPointGetInfo_AcpTrak_0();
	MC_BR_TrgPointGetInfo_AcpTrak_0.Execute := FALSE;
    // TON_0
	TON_0.PT := UDINT_TO_TIME(WaitTime);
	TON_0();
	// MC_BR_ShCopyUserData_AcpTrak
	MC_BR_ShCopyUserData_AcpTrak_0();
	MC_BR_ShCopyUserData_AcpTrak_0.Execute := FALSE;
	// MC_BR_RoutedMoveAbs_AcpTrak_0
	MC_BR_RoutedMoveAbs_AcpTrak_0.Sector 		  := SecAdr;
	MC_BR_RoutedMoveAbs_AcpTrak_0.Velocity		  := Speed_IN;
	MC_BR_RoutedMoveAbs_AcpTrak_0.Acceleration	  := Acc_IN;
	MC_BR_RoutedMoveAbs_AcpTrak_0.Deceleration	  := Acc_IN;
	MC_BR_RoutedMoveAbs_AcpTrak_0();
	MC_BR_RoutedMoveAbs_AcpTrak_0.Execute := FALSE;
	// MC_BR_ElasticMoveVel_AcpTrak_0
	MC_BR_ElasticMoveVel_AcpTrak_0.Velocity       := Speed_OUT;
	MC_BR_ElasticMoveVel_AcpTrak_0.Acceleration   := Acc_OUT;
	MC_BR_ElasticMoveVel_AcpTrak_0.Deceleration   := Acc_OUT;
	MC_BR_ElasticMoveVel_AcpTrak_0.Jerk           := 0.0;
	MC_BR_ElasticMoveVel_AcpTrak_0.Direction	  := mcDIR_POSITIVE;
	MC_BR_ElasticMoveVel_AcpTrak_0.BufferMode     := mcABORTING;
	MC_BR_ElasticMoveVel_AcpTrak_0();
	MC_BR_ElasticMoveVel_AcpTrak_0.Execute := FALSE;
	// MC_ReadStatus
	MC_ReadStatus_0();
	MC_ReadStatus_1();
	//MC_BR_BarrierCommand_AcpTrak
	MC_BR_BarrierCommand_AcpTrak_0();
	//MC_BR_BarrierReadInfo_AcpTrak
	MC_BR_BarrierReadInfo_AcpTrak_0.ProcessPoint := PPAdr;
	MC_BR_BarrierReadInfo_AcpTrak_0.Enable		 := TRUE;
	MC_BR_BarrierReadInfo_AcpTrak_0();

END_PROGRAM
```

### Program Logical/Source/ProcessTemplate/SingleSh/ProcStop_S3 (IEC) - trak process - 3 shuttles wait predefined time

#### Types.typ
```iecst
(*enum*)

TYPE
	StepEnum :
		(
		CHECK_TRIGGER,
		GET_SHUTTLE_DATA,
		GET_SHUTTLE_DATA_WAIT,
		GO_TO_PROCESS_STATION_1,
		GO_TO_PROCESS_STATION_2,
		GO_TO_PROCESS_STATION_3,
		GO_TO_PROCESS_STATION_WAIT,
		WAIT,
		SET_SHUTTLE_DATA,
		SET_SHUTTLE_DATA_WAIT,
		GO_TO_NEXT_STATION
		);
	StepTicket :
		(
		ENABLE_BARRIER := 0,
		OPENED_BARRIER,
		FREE_SHUTTLES
		);
END_TYPE
```

#### Variables.var
```iecst
(*process configuration*)
VAR
	PPAdr : UDINT;
	SecAdr : UDINT;
END_VAR
(*commands*)
VAR
	CmdEnableProcess : BOOL;
END_VAR
(*sequence control*)
VAR
	Step : StepEnum;
	ShuttleAxis : ARRAY[1..3] OF McAxisType;
	ShuttleUserData : ARRAY[1..3] OF TrakShuttleUserDataType;
	WaitTime : UDINT := 500;
	ProcPointPos : LREAL;
	CntShuttle : USINT;
	DistTravelled_1 : LREAL;
	DistTravelled_2 : LREAL;
	DistTravelled_3 : LREAL;
	ReleaseSts : BOOL;
END_VAR
(*barrier functionality*)
VAR
	sTickets : StepTicket; (*step variable for state machine*)
	cmdFreeShuttles : BOOL; (*When should the shuttles be released*)
END_VAR
(*colour configuration*)
VAR
	Red : REAL;
	Green : REAL;
	Blue : REAL;
END_VAR
(*movement configuration*)
VAR
	Speed_IN : REFERENCE TO REAL;
	Acc_IN : REFERENCE TO REAL;
	Speed_OUT : REFERENCE TO REAL;
	Acc_OUT : REFERENCE TO REAL;
END_VAR
(*FUB - Generic*)
VAR
	MC_BR_AsmReadStatus_AcpTrak_0 : MC_BR_AsmReadStatus_AcpTrak;
	MC_BR_TrgPointEnable_AcpTrak_0 : MC_BR_TrgPointEnable_AcpTrak;
	MC_BR_TrgPointGetInfo_AcpTrak_0 : MC_BR_TrgPointGetInfo_AcpTrak;
	MC_BR_ShCopyUserData_AcpTrak_0 : MC_BR_ShCopyUserData_AcpTrak;
	MC_BR_RoutedMoveAbs_AcpTrak_0 : MC_BR_RoutedMoveAbs_AcpTrak;
	MC_BR_ElasticMoveVel_AcpTrak_0 : MC_BR_ElasticMoveVel_AcpTrak;
	MC_BR_ProcPointGetInfo_AcpTrak_0 : MC_BR_ProcPointGetInfo_AcpTrak;
	MC_ReadStatus_0 : MC_ReadStatus;
	MC_ReadStatus_1 : MC_ReadStatus;
	MC_ReadStatus_2 : MC_ReadStatus;
	TON_0 : TON;
END_VAR
(*FUB - Barrier*)
VAR
	MC_BR_BarrierCommand_AcpTrak_0 : MC_BR_BarrierCommand_AcpTrak;
	MC_BR_BarrierReadInfo_AcpTrak_0 : MC_BR_BarrierReadInfo_AcpTrak;
END_VAR
```

#### Main.st
```iecst
(*********************************************************************************
 * Copyright: 	B&R Industrial Automation GmbH
 * Author:    	B&R ES
 * Created:   	April 8, 2022/10:54 AM
 * Description:	Three shuttles will be stopped a predefined time in the process
				station.
 * Mandatory: 	NO
 *********************************************************************************)
PROGRAM _INIT

	(*******************************************************************)
	(******************* Process Configuration *************************)
	(*******************************************************************)
	PPAdr 	:= ADR(PP_Test); 		// <-- NAME A VALID PROCESS POINT
	SecAdr	:= ADR(SectorTrackA);	// <-- NAME A VALID SECTOR
	(*** Define in/out speed & acceleration for this process ***)
	// IN
	Speed_IN ACCESS	ADR(gSpeedEmpty); 	// <-- Bind it to Empty / Full speed global variable
	Acc_IN ACCESS ADR(gAccEmpty); 		// <-- Bind it to Empty / Full acceleration global variable
	// OUT
	Speed_OUT ACCESS ADR(gSpeedFull); 	// <-- Bind it to Empty / Full speed global variable
	Acc_OUT	ACCESS ADR(gAccFull); 		// <-- Bind it to Empty / Full acceleration global variable
	(*** Define Wait Time (ms) ***)
	WaitTime := 500;
	(*** Define relative center point distance for the first coupled shuttles ***)
	DistTravelled_1	:= 0.99;
	DistTravelled_2 := 0.66;
	DistTravelled_3 := 0.33;
	(*** Define if it is a release station ***)
	ReleaseSts := FALSE;
	(*** SceneViewer - Shuttle color after process ***)
	Red	  := 0.02;
	Green := 0.77;
	Blue  := 0.21;
	(********************************************************************)

	CmdEnableProcess 	:= TRUE;
	cmdFreeShuttles		:= TRUE;
	Step 				:= CHECK_TRIGGER;

	MC_BR_ProcPointGetInfo_AcpTrak_0.ProcessPoint   := PPAdr;
	MC_BR_ProcPointGetInfo_AcpTrak_0.Execute		:= TRUE;

	REPEAT
		MC_BR_ProcPointGetInfo_AcpTrak_0();
	UNTIL
		MC_BR_ProcPointGetInfo_AcpTrak_0.Done OR MC_BR_ProcPointGetInfo_AcpTrak_0.Error
	END_REPEAT;

	ProcPointPos 	:= MC_BR_ProcPointGetInfo_AcpTrak_0.ProcPointInfo.SectorPosition.Position;
	CntShuttle 		:= 1;

END_PROGRAM

PROGRAM _CYCLIC

	///////////////// HIGH PRIORITY /////////////////
	(* reset process sequence if assembly is disabled *)
	IF EDGEPOS(gTrakAsm.StatusDisabled) THEN
		CntShuttle 		:= 1;
		TON_0.IN		:= FALSE;
		cmdFreeShuttles	:= (MC_BR_BarrierReadInfo_AcpTrak_0.BarrierInfo.RemainingTickets = 0);
		Step 			:= CHECK_TRIGGER;
	END_IF

	///////////// BARRIER FUNCTIONALITY /////////////
	(* this state machine is developed in such a way that allows to enable/disable the station without having to stop *)
	CASE sTickets OF
		ENABLE_BARRIER:
			MC_BR_BarrierCommand_AcpTrak_0.ProcessPoint := PPAdr;
			IF CmdEnableProcess THEN
				MC_BR_BarrierCommand_AcpTrak_0.Command := mcACPTRAK_BARRIER_CLOSE;
			ELSE
				MC_BR_BarrierCommand_AcpTrak_0.Command := mcACPTRAK_BARRIER_OPEN;
			END_IF
			MC_BR_BarrierCommand_AcpTrak_0.Execute := TRUE;
			IF (MC_BR_BarrierCommand_AcpTrak_0.Done) THEN
				MC_BR_BarrierCommand_AcpTrak_0.Execute := FALSE;
				IF CmdEnableProcess THEN
					sTickets := FREE_SHUTTLES;
				ELSE
					sTickets := OPENED_BARRIER;
				END_IF
			END_IF
		OPENED_BARRIER:
			IF EDGEPOS(CmdEnableProcess) THEN
				cmdFreeShuttles := (MC_BR_BarrierReadInfo_AcpTrak_0.BarrierInfo.RemainingTickets = 0);
				sTickets 		:= ENABLE_BARRIER;
			END_IF
		FREE_SHUTTLES:
			IF cmdFreeShuttles THEN
				MC_BR_BarrierCommand_AcpTrak_0.Command 							:= mcACPTRAK_BARRIER_ADD_TICKETS;
				MC_BR_BarrierCommand_AcpTrak_0.AdvancedParameters.TicketCount 	:= 1;
				MC_BR_BarrierCommand_AcpTrak_0.Execute 							:= TRUE;
				IF (MC_BR_BarrierCommand_AcpTrak_0.Done) THEN
					MC_BR_BarrierCommand_AcpTrak_0.Execute := FALSE;
					cmdFreeShuttles := FALSE;
				END_IF
			END_IF
			IF EDGENEG(CmdEnableProcess) THEN
				sTickets := ENABLE_BARRIER;
			END_IF
	END_CASE

	(***********************************************************************)
	(************************* STATE MACHINE *******************************)
	(***********************************************************************)

	CASE Step OF

		(* enable trigger and wait for one shuttle to pass *)
		CHECK_TRIGGER:
			IF((CmdEnableProcess) AND (MC_BR_AsmReadStatus_AcpTrak_0.AssemblyReady))THEN
				MC_BR_TrgPointEnable_AcpTrak_0.ProcessPoint  := PPAdr;
				MC_BR_TrgPointEnable_AcpTrak_0.Enable        := TRUE;
				(* shuttle passed => get axis reference *)
				IF((MC_BR_TrgPointEnable_AcpTrak_0.Valid) AND (MC_BR_TrgPointEnable_AcpTrak_0.EventCount > 0))THEN
					MC_BR_TrgPointGetInfo_AcpTrak_0.ProcessPoint  := PPAdr;
					MC_BR_TrgPointGetInfo_AcpTrak_0.Execute       := TRUE;
					Step := GET_SHUTTLE_DATA;
				END_IF
			ELSE
				MC_BR_TrgPointEnable_AcpTrak_0.Enable  := FALSE;
			END_IF

		(* axis reference of passed shuttle available *)
		(* get shuttle-UserData *)
		GET_SHUTTLE_DATA:

			IF(MC_BR_TrgPointGetInfo_AcpTrak_0.Done)THEN
				ShuttleAxis[CntShuttle] := MC_BR_TrgPointGetInfo_AcpTrak_0.TrgPointInfo.Axis;
				// read UserData from shuttle
				MC_BR_ShCopyUserData_AcpTrak_0.Axis         := ADR(ShuttleAxis[CntShuttle]);
				MC_BR_ShCopyUserData_AcpTrak_0.Execute      := TRUE;
				MC_BR_ShCopyUserData_AcpTrak_0.DataAddress  := ADR(ShuttleUserData[CntShuttle]);
				MC_BR_ShCopyUserData_AcpTrak_0.DataSize     := SIZEOF(ShuttleUserData[CntShuttle]);
				MC_BR_ShCopyUserData_AcpTrak_0.Mode         := mcACPTRAK_USERDATA_GET;
				Step := GET_SHUTTLE_DATA_WAIT;
			END_IF

		(* wait for shuttle-UserData content available *)
		GET_SHUTTLE_DATA_WAIT:
			IF(MC_BR_ShCopyUserData_AcpTrak_0.Done)THEN
				IF ShuttleUserData[CntShuttle].InitDone THEN
					CASE CntShuttle OF
						//First shuttle
						1:
							Step := GO_TO_PROCESS_STATION_1;
						// Second shuttle
						2:
							Step := GO_TO_PROCESS_STATION_2;
						// Third shuttle
						3:
							Step := GO_TO_PROCESS_STATION_3;
					END_CASE
				ELSE
					cmdFreeShuttles := (MC_BR_BarrierReadInfo_AcpTrak_0.BarrierInfo.RemainingTickets = 0);
					Step 			:= CHECK_TRIGGER;
				END_IF
			END_IF

		GO_TO_PROCESS_STATION_1:

			MC_BR_RoutedMoveAbs_AcpTrak_0.Axis			:= ADR(ShuttleAxis[CntShuttle]);
			MC_BR_RoutedMoveAbs_AcpTrak_0.Position 		:= ProcPointPos + DistTravelled_1;
			MC_BR_RoutedMoveAbs_AcpTrak_0.Execute 		:= TRUE;

			CntShuttle 		:= CntShuttle + 1;
			cmdFreeShuttles := TRUE;
			Step 			:= CHECK_TRIGGER;

		GO_TO_PROCESS_STATION_2:

			MC_BR_RoutedMoveAbs_AcpTrak_0.Axis			:= ADR(ShuttleAxis[CntShuttle]);
			MC_BR_RoutedMoveAbs_AcpTrak_0.Position 		:= ProcPointPos + DistTravelled_2;
			MC_BR_RoutedMoveAbs_AcpTrak_0.Execute 		:= TRUE;

			CntShuttle 		:= CntShuttle + 1;
			cmdFreeShuttles := TRUE;
			Step 			:= CHECK_TRIGGER;

		GO_TO_PROCESS_STATION_3:

			MC_BR_RoutedMoveAbs_AcpTrak_0.Axis			:= ADR(ShuttleAxis[CntShuttle]);
			MC_BR_RoutedMoveAbs_AcpTrak_0.Position 		:= ProcPointPos + DistTravelled_3;
			MC_BR_RoutedMoveAbs_AcpTrak_0.Execute 		:= TRUE;

			Step 		:= GO_TO_PROCESS_STATION_WAIT;

		GO_TO_PROCESS_STATION_WAIT:

			MC_ReadStatus_0.Axis 	:= ADR(ShuttleAxis[1]);
			MC_ReadStatus_0.Enable	:= TRUE;

			MC_ReadStatus_1.Axis 	:= ADR(ShuttleAxis[2]);
			MC_ReadStatus_1.Enable	:= TRUE;

			MC_ReadStatus_2.Axis 	:= ADR(ShuttleAxis[3]);
			MC_ReadStatus_2.Enable	:= TRUE;

			IF (MC_ReadStatus_0.StandStill AND MC_ReadStatus_1.StandStill AND MC_ReadStatus_2.StandStill) THEN
				MC_ReadStatus_0.Enable := FALSE;
				MC_ReadStatus_1.Enable := FALSE;
				MC_ReadStatus_2.Enable := FALSE;
				TON_0.IN 	:= TRUE;
				Step 		:= WAIT;
			END_IF

			IF (MC_BR_RoutedMoveAbs_AcpTrak_0.Done) THEN
				TON_0.IN 	:= TRUE;
				Step 		:= WAIT;
			END_IF

		WAIT:

			IF TON_0.Q THEN
				TON_0.IN 	:= FALSE;
				CntShuttle 	:= 1;
				Step 		:= SET_SHUTTLE_DATA;
			END_IF

		(* write modified UserData back to shuttle *)
		SET_SHUTTLE_DATA:

			ShuttleUserData[CntShuttle].SceneColorRed	:= Red;
			ShuttleUserData[CntShuttle].SceneColorGreen	:= Green;
			ShuttleUserData[CntShuttle].SceneColorBlue 	:= Blue;

			MC_BR_ShCopyUserData_AcpTrak_0.Axis         := ADR(ShuttleAxis[CntShuttle]);
			MC_BR_ShCopyUserData_AcpTrak_0.Execute      := TRUE;
			MC_BR_ShCopyUserData_AcpTrak_0.DataAddress  := ADR(ShuttleUserData[CntShuttle]);
			MC_BR_ShCopyUserData_AcpTrak_0.DataSize     := SIZEOF(ShuttleUserData[CntShuttle]);
			MC_BR_ShCopyUserData_AcpTrak_0.Mode         := mcACPTRAK_USERDATA_SET;
			Step := SET_SHUTTLE_DATA_WAIT;

		(* wait for shuttle-UserData content set *)
		SET_SHUTTLE_DATA_WAIT:

			IF(MC_BR_ShCopyUserData_AcpTrak_0.Done)THEN
				Step := GO_TO_NEXT_STATION;
			END_IF

			(* go to next station *)
		GO_TO_NEXT_STATION:

			MC_BR_ElasticMoveVel_AcpTrak_0.Axis           := ADR(ShuttleAxis[CntShuttle]);
			MC_BR_ElasticMoveVel_AcpTrak_0.Execute        := TRUE;

			IF ReleaseSts THEN
				gProducedProduct := gProducedProduct + 3;
			END_IF

			CASE CntShuttle OF
				1..2:
					CntShuttle 	:= CntShuttle + 1;
					Step		:= SET_SHUTTLE_DATA;
				3:
					CntShuttle		:= 1;
					cmdFreeShuttles := TRUE;
					Step 			:= CHECK_TRIGGER;
			END_CASE

	END_CASE

	(*** Call all function blocks ***)
	// MC_BR_AsmReadStatus_AcpTrak
	MC_BR_AsmReadStatus_AcpTrak_0.Assembly 	:= ADR(gAssembly_1);
	MC_BR_AsmReadStatus_AcpTrak_0.Enable 	:= TRUE;
	MC_BR_AsmReadStatus_AcpTrak_0();
    // MC_BR_TrgPointEnable_AcpTrak
	MC_BR_TrgPointEnable_AcpTrak_0();
    // MC_BR_TrgPointGetInfo_AcpTrak
	MC_BR_TrgPointGetInfo_AcpTrak_0();
	MC_BR_TrgPointGetInfo_AcpTrak_0.Execute := FALSE;
    // TON_0
	TON_0.PT := UDINT_TO_TIME(WaitTime);
	TON_0();
	// MC_BR_ShCopyUserData_AcpTrak
	MC_BR_ShCopyUserData_AcpTrak_0();
	MC_BR_ShCopyUserData_AcpTrak_0.Execute := FALSE;
	// MC_BR_RoutedMoveAbs_AcpTrak_0
	MC_BR_RoutedMoveAbs_AcpTrak_0.Sector 		  := SecAdr;
	MC_BR_RoutedMoveAbs_AcpTrak_0.Velocity		  := Speed_IN;
	MC_BR_RoutedMoveAbs_AcpTrak_0.Acceleration	  := Acc_IN;
	MC_BR_RoutedMoveAbs_AcpTrak_0.Deceleration	  := Acc_IN;
	MC_BR_RoutedMoveAbs_AcpTrak_0();
	MC_BR_RoutedMoveAbs_AcpTrak_0.Execute := FALSE;
	// MC_BR_ElasticMoveVel_AcpTrak_0
	MC_BR_ElasticMoveVel_AcpTrak_0.Velocity       := Speed_OUT;
	MC_BR_ElasticMoveVel_AcpTrak_0.Acceleration   := Acc_OUT;
	MC_BR_ElasticMoveVel_AcpTrak_0.Deceleration   := Acc_OUT;
	MC_BR_ElasticMoveVel_AcpTrak_0.Jerk           := 0.0;
	MC_BR_ElasticMoveVel_AcpTrak_0.Direction	  := mcDIR_POSITIVE;
	MC_BR_ElasticMoveVel_AcpTrak_0.BufferMode     := mcABORTING;
	MC_BR_ElasticMoveVel_AcpTrak_0();
	MC_BR_ElasticMoveVel_AcpTrak_0.Execute := FALSE;
	// MC_ReadStatus
	MC_ReadStatus_0();
	MC_ReadStatus_1();
	MC_ReadStatus_2();
	//MC_BR_BarrierCommand_AcpTrak
	MC_BR_BarrierCommand_AcpTrak_0();
	//MC_BR_BarrierReadInfo_AcpTrak
	MC_BR_BarrierReadInfo_AcpTrak_0.ProcessPoint := PPAdr;
	MC_BR_BarrierReadInfo_AcpTrak_0.Enable		 := TRUE;
	MC_BR_BarrierReadInfo_AcpTrak_0();

END_PROGRAM
```

### Package Logical/Source/ProcessTemplate/PairedSh - paired shuttle operation

### Program Logical/Source/ProcessTemplate/PairedSh/ProcSync (IEC) - trak process - sync. between 2 shuttles

#### Types.typ
```iecst
(*enum*)

TYPE
	StepEnum :
		(
		CHECK_TRIGGER := 0,
		GET_USERDATA,
		GO_TO_SYNC_POS,
		GO_TO_SYNC_POS_WAIT,
		CREATE_CONV,
		CREATE_CONV_WAIT,
		ADD_SH_CONV,
		ADD_SH_CONV_WAIT,
		SET_USERDATA,
		SET_USERDATA_WAIT,
		GO_TO_NEXT_STATION
		);
END_TYPE
```

#### Variables.var
```iecst
(*process configuration*)
VAR
	PPAdr : UDINT;
	SecAdr : UDINT;
END_VAR
(*commands*)
VAR
	CmdEnableProcess : BOOL;
END_VAR
(*sequence control*)
VAR
	Step : StepEnum;
	ShuttleAxis : ARRAY[1..2] OF McAxisType;
	ShuttleUserData : ARRAY[1..2] OF TrakShuttleUserDataType;
	CntShuttle : USINT;
	ProcPointPos : LREAL;
END_VAR
(*colour configuration*)
VAR
	Red : REAL;
	Green : REAL;
	Blue : REAL;
END_VAR
(*movement configuration*)
VAR
	Speed_IN : REFERENCE TO REAL;
	Acc_IN : REFERENCE TO REAL;
	Speed_OUT : REFERENCE TO REAL;
	Acc_OUT : REFERENCE TO REAL;
END_VAR
(*process-point FUB*)
VAR
	MC_BR_TrgPointEnable_AcpTrak_0 : MC_BR_TrgPointEnable_AcpTrak;
	MC_BR_TrgPointGetInfo_AcpTrak_0 : MC_BR_TrgPointGetInfo_AcpTrak;
	MC_BR_ShCopyUserData_AcpTrak_0 : MC_BR_ShCopyUserData_AcpTrak;
	MC_BR_BarrierCommand_AcpTrak_0 : MC_BR_BarrierCommand_AcpTrak;
	MC_BR_BarrierReadInfo_AcpTrak_0 : MC_BR_BarrierReadInfo_AcpTrak;
	MC_BR_ShCreateConvoy_AcpTrak_0 : MC_BR_ShCreateConvoy_AcpTrak;
	MC_BR_ShMoveInConvoy_AcpTrak_0 : MC_BR_ShMoveInConvoy_AcpTrak;
	MC_BR_ProcPointGetInfo_AcpTrak_0 : MC_BR_ProcPointGetInfo_AcpTrak;
	MC_BR_RoutedMoveAbs_AcpTrak_0 : MC_BR_RoutedMoveAbs_AcpTrak;
	MC_BR_ElasticMoveVel_AcpTrak_0 : MC_BR_ElasticMoveVel_AcpTrak;
END_VAR
```

#### Main.st
```iecst
(*********************************************************************************
 * Copyright: 	B&R Industrial Automation GmbH
 * Author:    	B&R ES
 * Created:   	April 8, 2022/10:54 AM
 * Description:	All the shuttles crossing this process point will be synched and
				initialized.
 * Mandatory: 	YES - Should be allways included before paired shuttle station
				operations.
 *********************************************************************************)
PROGRAM _INIT

	(*******************************************************************)
	(******************* Process Configuration *************************)
	(*******************************************************************)
	PPAdr 	:= ADR(PP_Test); 		// <-- NAME A VALID PROCESS POINT
	SecAdr	:= ADR(SectorTrackA);	// <-- NAME A VALID SECTOR
	(*** Define in/out speed & acceleration for this process ***)
	// IN
	Speed_IN ACCESS	ADR(gSpeedEmpty); 	// <-- Bind it to Empty / Full speed global variable
	Acc_IN ACCESS ADR(gAccEmpty); 		// <-- Bind it to Empty / Full acceleration global variable
	// OUT
	Speed_OUT ACCESS ADR(gSpeedFull); 	// <-- Bind it to Empty / Full speed global variable
	Acc_OUT	ACCESS ADR(gAccFull); 		// <-- Bind it to Empty / Full acceleration global variable
	(*** SceneViewer - Shuttle color after process ***)
	Red	  := 0.0;
	Green := 1.0;
	Blue  := 0.0;
	(********************************************************************)

	(* Local variable to enable/disable the process *)
	CmdEnableProcess := TRUE;

	(* Processpointreference for Functionblocks *)
	MC_BR_TrgPointEnable_AcpTrak_0.ProcessPoint 	:= PPAdr;
	MC_BR_TrgPointGetInfo_AcpTrak_0.ProcessPoint 	:= PPAdr;

	(* Barrier configuration *)
	// Barrier command
	MC_BR_BarrierCommand_AcpTrak_0.ProcessPoint 					:= PPAdr;
	MC_BR_BarrierCommand_AcpTrak_0.Command 							:= mcACPTRAK_BARRIER_ADD_TICKETS;
	MC_BR_BarrierCommand_AcpTrak_0.AdvancedParameters.TicketCount 	:= 1;
	MC_BR_BarrierCommand_AcpTrak_0.Execute 							:= TRUE; (* To initialize the barrier *)

	(* Get process point position *)
	MC_BR_ProcPointGetInfo_AcpTrak_0.ProcessPoint   := PPAdr;
	MC_BR_ProcPointGetInfo_AcpTrak_0.Execute		:= TRUE;

	REPEAT
		MC_BR_ProcPointGetInfo_AcpTrak_0();
		UNTIL
		MC_BR_ProcPointGetInfo_AcpTrak_0.Done OR MC_BR_ProcPointGetInfo_AcpTrak_0.Error
	END_REPEAT;

	ProcPointPos 	:= MC_BR_ProcPointGetInfo_AcpTrak_0.ProcPointInfo.SectorPosition.Position;

	(* Counting variable *)
	CntShuttle := 1;

END_PROGRAM

PROGRAM _CYCLIC

	//////////////////// HIGH PRIORITY ///////////////////
	IF gTrakAsm.StatusDisabled THEN
		CntShuttle 	:= 1;
		IF (MC_BR_BarrierReadInfo_AcpTrak_0.BarrierInfo.RemainingTickets = 0) AND (MC_BR_BarrierReadInfo_AcpTrak_0.Valid) THEN
			MC_BR_BarrierCommand_AcpTrak_0.Execute := TRUE;
		END_IF
		Step 		:= CHECK_TRIGGER;
	END_IF
	//////////////////////////////////////////////////////

	CASE Step OF

		CHECK_TRIGGER:

			(* When the process is enabled and the assembly is ready, the process will be activated *)
			IF((CmdEnableProcess) AND (gTrakAsm.StatusReady))THEN
				MC_BR_TrgPointEnable_AcpTrak_0.Enable := TRUE;
				(* If a shuttle passes the triggerpoint then get the axis reference *)
				IF((MC_BR_TrgPointEnable_AcpTrak_0.Valid) AND (MC_BR_TrgPointEnable_AcpTrak_0.EventCount > 0))THEN
					MC_BR_TrgPointGetInfo_AcpTrak_0.Execute := TRUE;
				END_IF
			ELSE
				(* Else the processpoint will be disabled *)
				MC_BR_TrgPointEnable_AcpTrak_0.Enable := FALSE;
			END_IF

			(* If axis reference is available, save it and go to the next step *)
			IF EDGEPOS(MC_BR_TrgPointGetInfo_AcpTrak_0.Done) THEN
			(* Save axis reference in local variable for use in step machine *)
				ShuttleAxis[CntShuttle]	:= MC_BR_TrgPointGetInfo_AcpTrak_0.TrgPointInfo.Axis;
				Step := GET_USERDATA;
			END_IF

		GET_USERDATA:

			(* The userdata is copied on a local variable *)
			MC_BR_ShCopyUserData_AcpTrak_0.Axis 		:= ADR(ShuttleAxis[CntShuttle]);
			MC_BR_ShCopyUserData_AcpTrak_0.Execute 		:= TRUE;
			MC_BR_ShCopyUserData_AcpTrak_0.DataAddress	:= ADR(ShuttleUserData[CntShuttle]);
			MC_BR_ShCopyUserData_AcpTrak_0.DataSize 	:= SIZEOF(ShuttleUserData[CntShuttle]);
			MC_BR_ShCopyUserData_AcpTrak_0.Mode 		:= mcACPTRAK_USERDATA_GET;
			(* After copying go to the next step *)
			IF EDGEPOS(MC_BR_ShCopyUserData_AcpTrak_0.Done) THEN
				Step := GO_TO_SYNC_POS;
			END_IF

		GO_TO_SYNC_POS:

			MC_BR_RoutedMoveAbs_AcpTrak_0.Axis 	:= ADR(ShuttleAxis[CntShuttle]);
			MC_BR_RoutedMoveAbs_AcpTrak_0.Execute	:= TRUE;

			IF CntShuttle = 1 THEN
				MC_BR_RoutedMoveAbs_AcpTrak_0.Position := ProcPointPos + 0.05 + gProductWidth;
			ELSE
				MC_BR_RoutedMoveAbs_AcpTrak_0.Position := ProcPointPos + 0.05;
			END_IF

			Step := GO_TO_SYNC_POS_WAIT;

		GO_TO_SYNC_POS_WAIT:

			IF MC_BR_RoutedMoveAbs_AcpTrak_0.Done THEN
				IF CntShuttle = 1 THEN
					CntShuttle 	:= CntShuttle + 1;
					Step 		:= CREATE_CONV;
				ELSE
					Step 		:= ADD_SH_CONV;
				END_IF
			END_IF

		CREATE_CONV:

			(* Creates the convoy adding a master shuttle *)
			MC_BR_ShCreateConvoy_AcpTrak_0.Axis 		:= ADR(ShuttleAxis[1]);
			MC_BR_ShCreateConvoy_AcpTrak_0.Execute		:= TRUE;
			Step := CREATE_CONV_WAIT;

		CREATE_CONV_WAIT:

			IF MC_BR_ShCreateConvoy_AcpTrak_0.Done THEN
				MC_BR_BarrierCommand_AcpTrak_0.Execute := TRUE;
				Step := CHECK_TRIGGER;
			END_IF

		ADD_SH_CONV:

			(* Add one shuttle to the convoy *)
			MC_BR_ShMoveInConvoy_AcpTrak_0.Axis							:= ADR(ShuttleAxis[2]);
			MC_BR_ShMoveInConvoy_AcpTrak_0.Execute						:= TRUE;
			MC_BR_ShMoveInConvoy_AcpTrak_0.Parameters.ReferenceShuttle 	:= ADR(ShuttleAxis[1]);

			Step := ADD_SH_CONV_WAIT;

		ADD_SH_CONV_WAIT:

			(* Wait until shuttke us added to the convoy *)
			IF MC_BR_ShMoveInConvoy_AcpTrak_0.Done THEN
				CntShuttle 	:= 1;
				Step 		:= SET_USERDATA;
			END_IF

		SET_USERDATA:

			(* Change color to know that shuttles are in sync. *)
			ShuttleUserData[CntShuttle].SceneColorRed 	:= Red;
			ShuttleUserData[CntShuttle].SceneColorGreen := Green;
			ShuttleUserData[CntShuttle].SceneColorBlue	:= Blue;

			(* After this point, the shuttle is initialized *)
			ShuttleUserData[CntShuttle].InitDone := TRUE;

			(* The modified userdata will be copied back on the shuttle *)
			MC_BR_ShCopyUserData_AcpTrak_0.Axis 		:= ADR(ShuttleAxis[CntShuttle]);
			MC_BR_ShCopyUserData_AcpTrak_0.Execute 		:= TRUE;
			MC_BR_ShCopyUserData_AcpTrak_0.DataAddress	:= ADR(ShuttleUserData[CntShuttle]);
			MC_BR_ShCopyUserData_AcpTrak_0.DataSize 	:= SIZEOF(ShuttleUserData[CntShuttle]);
			MC_BR_ShCopyUserData_AcpTrak_0.Mode 		:= mcACPTRAK_USERDATA_SET;
			Step := SET_USERDATA_WAIT;

		SET_USERDATA_WAIT:

			IF (MC_BR_ShCopyUserData_AcpTrak_0.Done) THEN
				(* Move the second shuttle to the next station *)
				IF (CntShuttle = 1) THEN
					CntShuttle 	:= 2;
					Step 		:= SET_USERDATA;
				ELSE (* Let the next pair of shuttles in the station *)
					CntShuttle 	:= 1;
					Step 		:= GO_TO_NEXT_STATION;
				END_IF
			END_IF

		GO_TO_NEXT_STATION:

			MC_BR_ElasticMoveVel_AcpTrak_0.Axis 	:= ADR(ShuttleAxis[1]);
			MC_BR_ElasticMoveVel_AcpTrak_0.Execute	:= TRUE;

			MC_BR_BarrierCommand_AcpTrak_0.Execute  := TRUE;
			Step := CHECK_TRIGGER;

	END_CASE

	(*** Call all function blocks ***)
	// MC_BR_TrgPointEnable_AcpTrak
	MC_BR_TrgPointEnable_AcpTrak_0();
	// MC_BR_TrgPointGetInfo_AcpTrak
	MC_BR_TrgPointGetInfo_AcpTrak_0();
	MC_BR_TrgPointGetInfo_AcpTrak_0.Execute  := FALSE;
	// MC_BR_ShCopyUserData_AcpTrak
	MC_BR_ShCopyUserData_AcpTrak_0();
	MC_BR_ShCopyUserData_AcpTrak_0.Execute 	 := FALSE;
	// MC_BR_ShCreateConvoy_AcpTrak
	MC_BR_ShCreateConvoy_AcpTrak_0();
	MC_BR_ShCreateConvoy_AcpTrak_0.Execute := FALSE;
	// MC_BR_ShMoveInConvoy_AcpTrak
	MC_BR_ShMoveInConvoy_AcpTrak_0();
	MC_BR_ShMoveInConvoy_AcpTrak_0.Execute := FALSE;
	// MC_BR_BarrierCommand_AcpTrak
	MC_BR_BarrierCommand_AcpTrak_0();
	(* When adding tickets is done, reset the execute *)
	IF EDGEPOS(MC_BR_BarrierCommand_AcpTrak_0.Done) THEN
		MC_BR_BarrierCommand_AcpTrak_0.Execute := FALSE;
	END_IF
	// MC_BR_BarrierReadInfo_AcpTrak
	MC_BR_BarrierReadInfo_AcpTrak_0.ProcessPoint := PPAdr;
	MC_BR_BarrierReadInfo_AcpTrak_0.Enable 		 := TRUE;
	MC_BR_BarrierReadInfo_AcpTrak_0();
	// MC_BR_RoutedMoveAbs_AcpTrak_0
	MC_BR_RoutedMoveAbs_AcpTrak_0.Sector 		  := SecAdr;
	MC_BR_RoutedMoveAbs_AcpTrak_0.Velocity		  := Speed_IN;
	MC_BR_RoutedMoveAbs_AcpTrak_0.Acceleration	  := Acc_IN;
	MC_BR_RoutedMoveAbs_AcpTrak_0.Deceleration	  := Acc_IN;
	MC_BR_RoutedMoveAbs_AcpTrak_0();
	MC_BR_RoutedMoveAbs_AcpTrak_0.Execute := FALSE;
	// MC_BR_ElasticMoveVel_AcpTrak_0
	MC_BR_ElasticMoveVel_AcpTrak_0.Velocity       := Speed_OUT;
	MC_BR_ElasticMoveVel_AcpTrak_0.Acceleration   := Acc_OUT;
	MC_BR_ElasticMoveVel_AcpTrak_0.Deceleration   := Acc_OUT;
	MC_BR_ElasticMoveVel_AcpTrak_0.Jerk           := 0.0;
	MC_BR_ElasticMoveVel_AcpTrak_0.Direction	  := mcDIR_POSITIVE;
	MC_BR_ElasticMoveVel_AcpTrak_0.BufferMode     := mcABORTING;
	MC_BR_ElasticMoveVel_AcpTrak_0();
	MC_BR_ElasticMoveVel_AcpTrak_0.Execute := FALSE;

END_PROGRAM
```

- Main.st.bak (not shown)

### Program Logical/Source/ProcessTemplate/PairedSh/ProcUnSync (IEC) - trak process - unsync. shuttles

#### Types.typ
```iecst
(*enum*)

TYPE
	StepEnum :
		(
		CHECK_TRIGGER := 0,
		GET_USERDATA,
		SET_USERDATA,
		SET_USERDATA_WAIT,
		GO_TO_NEXT_STATION
		);
END_TYPE
```

#### Variables.var
```iecst
(*process configuration*)
VAR
	PPAdr : UDINT;
END_VAR
(*commands*)
VAR
	CmdEnableProcess : BOOL;
END_VAR
(*sequence control*)
VAR
	Step : StepEnum;
	ShuttleAxis : McAxisType;
	ShuttleUserData : TrakShuttleUserDataType;
END_VAR
(*colour configuration*)
VAR
	Red : REAL;
	Green : REAL;
	Blue : REAL;
END_VAR
(*movement configuration*)
VAR
	Speed_OUT : REFERENCE TO REAL;
	Acc_OUT : REFERENCE TO REAL;
END_VAR
(*process-point FUB*)
VAR
	MC_BR_TrgPointEnable_AcpTrak_0 : MC_BR_TrgPointEnable_AcpTrak;
	MC_BR_TrgPointGetInfo_AcpTrak_0 : MC_BR_TrgPointGetInfo_AcpTrak;
	MC_BR_ShCopyUserData_AcpTrak_0 : MC_BR_ShCopyUserData_AcpTrak;
	MC_BR_BarrierReadInfo_AcpTrak_0 : MC_BR_BarrierReadInfo_AcpTrak;
	MC_BR_ElasticMoveVel_AcpTrak_0 : MC_BR_ElasticMoveVel_AcpTrak;
END_VAR
```
